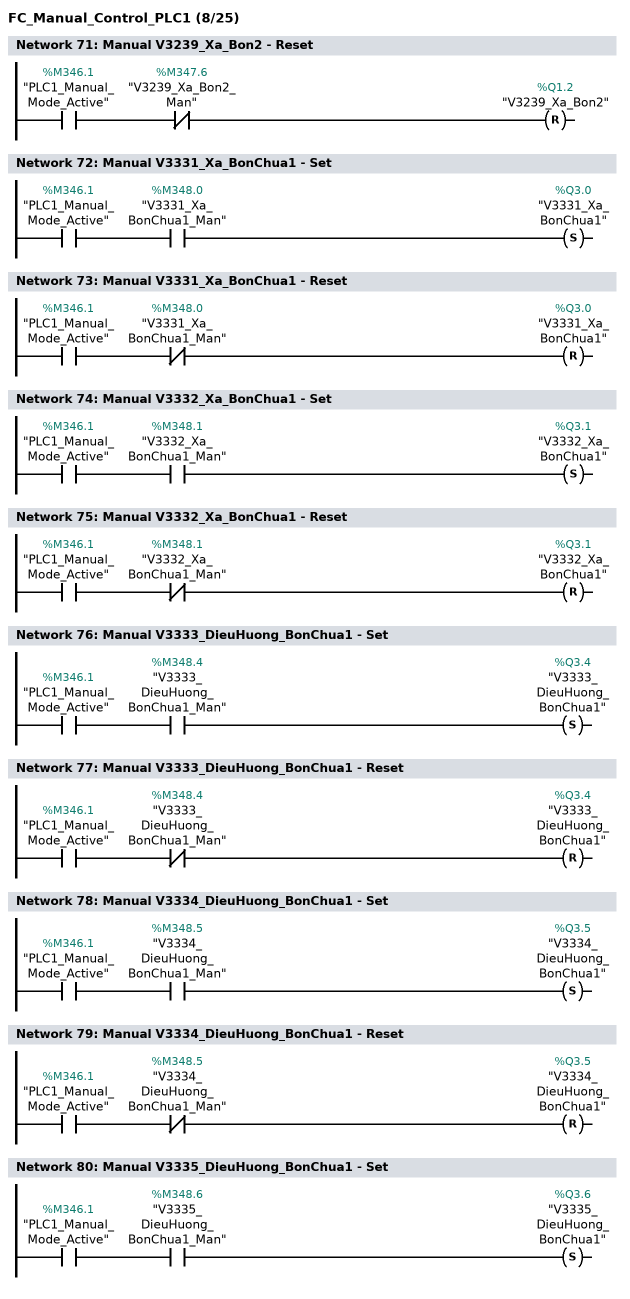
   RUNG wire#powerrail
      Contact( "PLC1_Manual_Mode_Active" )
      I_Contact( "V3239_Xa_Bon2_Man" )
      R_Coil( "V3239_Xa_Bon2" )
   END_RUNG
   // the same network as SCL:
   IF "PLC1_Manual_Mode_Active" AND NOT "V3239_Xa_Bon2_Man" THEN "V3239_Xa_Bon2" := FALSE; END_IF;
END_REGION

REGION Network 72: Manual V3331_Xa_BonChua1 - Set
   RUNG wire#powerrail
      Contact( "PLC1_Manual_Mode_Active" )
      Contact( "V3331_Xa_BonChua1_Man" )
      S_Coil( "V3331_Xa_BonChua1" )
   END_RUNG
   // the same network as SCL:
   IF "PLC1_Manual_Mode_Active" AND "V3331_Xa_BonChua1_Man" THEN "V3331_Xa_BonChua1" := TRUE; END_IF;
END_REGION

REGION Network 73: Manual V3331_Xa_BonChua1 - Reset
   RUNG wire#powerrail
      Contact( "PLC1_Manual_Mode_Active" )
      I_Contact( "V3331_Xa_BonChua1_Man" )
      R_Coil( "V3331_Xa_BonChua1" )
   END_RUNG
   // the same network as SCL:
   IF "PLC1_Manual_Mode_Active" AND NOT "V3331_Xa_BonChua1_Man" THEN "V3331_Xa_BonChua1" := FALSE; END_IF;
END_REGION

REGION Network 74: Manual V3332_Xa_BonChua1 - Set
   RUNG wire#powerrail
      Contact( "PLC1_Manual_Mode_Active" )
      Contact( "V3332_Xa_BonChua1_Man" )
      S_Coil( "V3332_Xa_BonChua1" )
   END_RUNG
   // the same network as SCL:
   IF "PLC1_Manual_Mode_Active" AND "V3332_Xa_BonChua1_Man" THEN "V3332_Xa_BonChua1" := TRUE; END_IF;
END_REGION

REGION Network 75: Manual V3332_Xa_BonChua1 - Reset
   RUNG wire#powerrail
      Contact( "PLC1_Manual_Mode_Active" )
      I_Contact( "V3332_Xa_BonChua1_Man" )
      R_Coil( "V3332_Xa_BonChua1" )
   END_RUNG
   // the same network as SCL:
   IF "PLC1_Manual_Mode_Active" AND NOT "V3332_Xa_BonChua1_Man" THEN "V3332_Xa_BonChua1" := FALSE; END_IF;
END_REGION

REGION Network 76: Manual V3333_DieuHuong_BonChua1 - Set
   RUNG wire#powerrail
      Contact( "PLC1_Manual_Mode_Active" )
      Contact( "V3333_DieuHuong_BonChua1_Man" )
      S_Coil( "V3333_DieuHuong_BonChua1" )
   END_RUNG
   // the same network as SCL:
   IF "PLC1_Manual_Mode_Active" AND "V3333_DieuHuong_BonChua1_Man" THEN
       "V3333_DieuHuong_BonChua1" := TRUE;
   END_IF;
END_REGION

REGION Network 77: Manual V3333_DieuHuong_BonChua1 - Reset
   RUNG wire#powerrail
      Contact( "PLC1_Manual_Mode_Active" )
      I_Contact( "V3333_DieuHuong_BonChua1_Man" )
      R_Coil( "V3333_DieuHuong_BonChua1" )
   END_RUNG
   // the same network as SCL:
   IF "PLC1_Manual_Mode_Active" AND NOT "V3333_DieuHuong_BonChua1_Man" THEN
       "V3333_DieuHuong_BonChua1" := FALSE;
   END_IF;
END_REGION

REGION Network 78: Manual V3334_DieuHuong_BonChua1 - Set
   RUNG wire#powerrail
      Contact( "PLC1_Manual_Mode_Active" )
      Contact( "V3334_DieuHuong_BonChua1_Man" )
      S_Coil( "V3334_DieuHuong_BonChua1" )
   END_RUNG
   // the same network as SCL:
   IF "PLC1_Manual_Mode_Active" AND "V3334_DieuHuong_BonChua1_Man" THEN
       "V3334_DieuHuong_BonChua1" := TRUE;
   END_IF;
END_REGION

REGION Network 79: Manual V3334_DieuHuong_BonChua1 - Reset
   RUNG wire#powerrail
      Contact( "PLC1_Manual_Mode_Active" )
      I_Contact( "V3334_DieuHuong_BonChua1_Man" )
      R_Coil( "V3334_DieuHuong_BonChua1" )
   END_RUNG
   // the same network as SCL:
   IF "PLC1_Manual_Mode_Active" AND NOT "V3334_DieuHuong_BonChua1_Man" THEN
       "V3334_DieuHuong_BonChua1" := FALSE;
   END_IF;
END_REGION

REGION Network 80: Manual V3335_DieuHuong_BonChua1 - Set
   RUNG wire#powerrail
      Contact( "PLC1_Manual_Mode_Active" )
      Contact( "V3335_DieuHuong_BonChua1_Man" )
      S_Coil( "V3335_DieuHuong_BonChua1" )
   END_RUNG
   // the same network as SCL:
   IF "PLC1_Manual_Mode_Active" AND "V3335_DieuHuong_BonChua1_Man" THEN
       "V3335_DieuHuong_BonChua1" := TRUE;
   END_IF;
END_REGION

REGION Network 81: Manual V3335_DieuHuong_BonChua1 - Reset
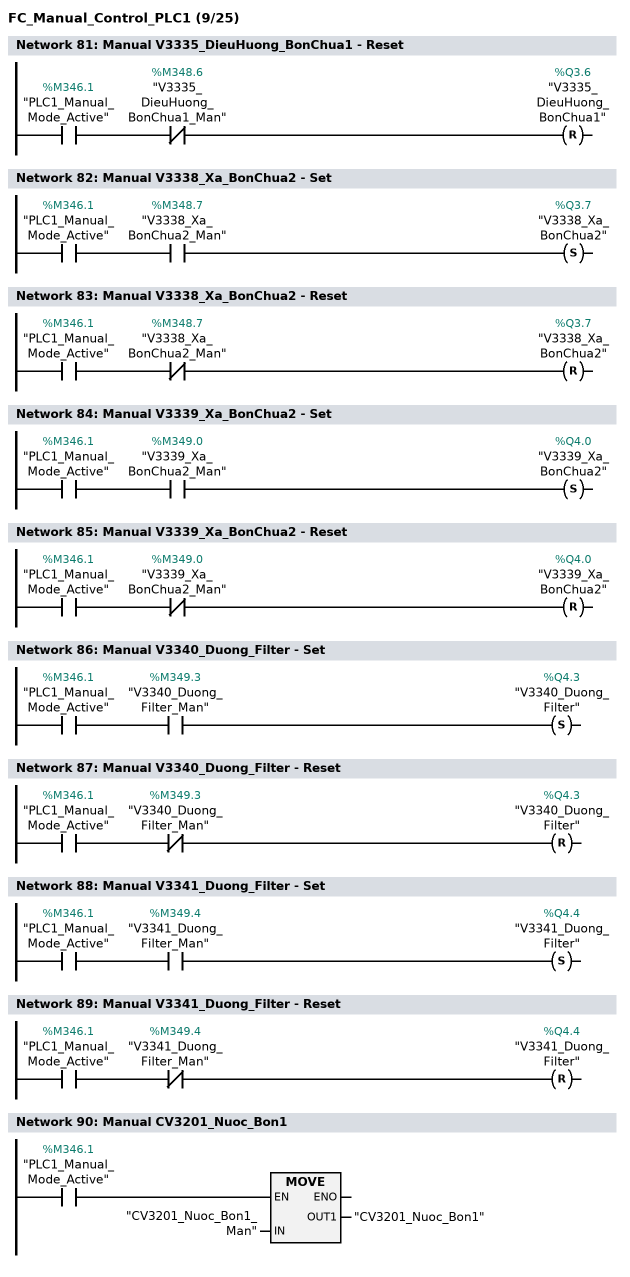
   RUNG wire#powerrail
      Contact( "PLC1_Manual_Mode_Active" )
      I_Contact( "V3335_DieuHuong_BonChua1_Man" )
      R_Coil( "V3335_DieuHuong_BonChua1" )
   END_RUNG
   // the same network as SCL:
   IF "PLC1_Manual_Mode_Active" AND NOT "V3335_DieuHuong_BonChua1_Man" THEN
       "V3335_DieuHuong_BonChua1" := FALSE;
   END_IF;
END_REGION

REGION Network 82: Manual V3338_Xa_BonChua2 - Set
   RUNG wire#powerrail
      Contact( "PLC1_Manual_Mode_Active" )
      Contact( "V3338_Xa_BonChua2_Man" )
      S_Coil( "V3338_Xa_BonChua2" )
   END_RUNG
   // the same network as SCL:
   IF "PLC1_Manual_Mode_Active" AND "V3338_Xa_BonChua2_Man" THEN "V3338_Xa_BonChua2" := TRUE; END_IF;
END_REGION

REGION Network 83: Manual V3338_Xa_BonChua2 - Reset
   RUNG wire#powerrail
      Contact( "PLC1_Manual_Mode_Active" )
      I_Contact( "V3338_Xa_BonChua2_Man" )
      R_Coil( "V3338_Xa_BonChua2" )
   END_RUNG
   // the same network as SCL:
   IF "PLC1_Manual_Mode_Active" AND NOT "V3338_Xa_BonChua2_Man" THEN "V3338_Xa_BonChua2" := FALSE; END_IF;
END_REGION

REGION Network 84: Manual V3339_Xa_BonChua2 - Set
   RUNG wire#powerrail
      Contact( "PLC1_Manual_Mode_Active" )
      Contact( "V3339_Xa_BonChua2_Man" )
      S_Coil( "V3339_Xa_BonChua2" )
   END_RUNG
   // the same network as SCL:
   IF "PLC1_Manual_Mode_Active" AND "V3339_Xa_BonChua2_Man" THEN "V3339_Xa_BonChua2" := TRUE; END_IF;
END_REGION

REGION Network 85: Manual V3339_Xa_BonChua2 - Reset
   RUNG wire#powerrail
      Contact( "PLC1_Manual_Mode_Active" )
      I_Contact( "V3339_Xa_BonChua2_Man" )
      R_Coil( "V3339_Xa_BonChua2" )
   END_RUNG
   // the same network as SCL:
   IF "PLC1_Manual_Mode_Active" AND NOT "V3339_Xa_BonChua2_Man" THEN "V3339_Xa_BonChua2" := FALSE; END_IF;
END_REGION

REGION Network 86: Manual V3340_Duong_Filter - Set
   RUNG wire#powerrail
      Contact( "PLC1_Manual_Mode_Active" )
      Contact( "V3340_Duong_Filter_Man" )
      S_Coil( "V3340_Duong_Filter" )
   END_RUNG
   // the same network as SCL:
   IF "PLC1_Manual_Mode_Active" AND "V3340_Duong_Filter_Man" THEN "V3340_Duong_Filter" := TRUE; END_IF;
END_REGION

REGION Network 87: Manual V3340_Duong_Filter - Reset
   RUNG wire#powerrail
      Contact( "PLC1_Manual_Mode_Active" )
      I_Contact( "V3340_Duong_Filter_Man" )
      R_Coil( "V3340_Duong_Filter" )
   END_RUNG
   // the same network as SCL:
   IF "PLC1_Manual_Mode_Active" AND NOT "V3340_Duong_Filter_Man" THEN "V3340_Duong_Filter" := FALSE; END_IF;
END_REGION

REGION Network 88: Manual V3341_Duong_Filter - Set
   RUNG wire#powerrail
      Contact( "PLC1_Manual_Mode_Active" )
      Contact( "V3341_Duong_Filter_Man" )
      S_Coil( "V3341_Duong_Filter" )
   END_RUNG
   // the same network as SCL:
   IF "PLC1_Manual_Mode_Active" AND "V3341_Duong_Filter_Man" THEN "V3341_Duong_Filter" := TRUE; END_IF;
END_REGION

REGION Network 89: Manual V3341_Duong_Filter - Reset
   RUNG wire#powerrail
      Contact( "PLC1_Manual_Mode_Active" )
      I_Contact( "V3341_Duong_Filter_Man" )
      R_Coil( "V3341_Duong_Filter" )
   END_RUNG
   // the same network as SCL:
   IF "PLC1_Manual_Mode_Active" AND NOT "V3341_Duong_Filter_Man" THEN "V3341_Duong_Filter" := FALSE; END_IF;
END_REGION

REGION Network 90: Manual CV3201_Nuoc_Bon1
   RUNG wire#powerrail
      Contact( "PLC1_Manual_Mode_Active" )
      { S7_GenerateENO := "TRUE" } Move(in := "CV3201_Nuoc_Bon1_Man", out1 => "CV3201_Nuoc_Bon1")
   END_RUNG
   // the same network as SCL:
   IF "PLC1_Manual_Mode_Active" THEN "CV3201_Nuoc_Bon1" := "CV3201_Nuoc_Bon1_Man"; END_IF;
END_REGION

REGION Network 91: Manual AGTR3260_Toc_Do_AO
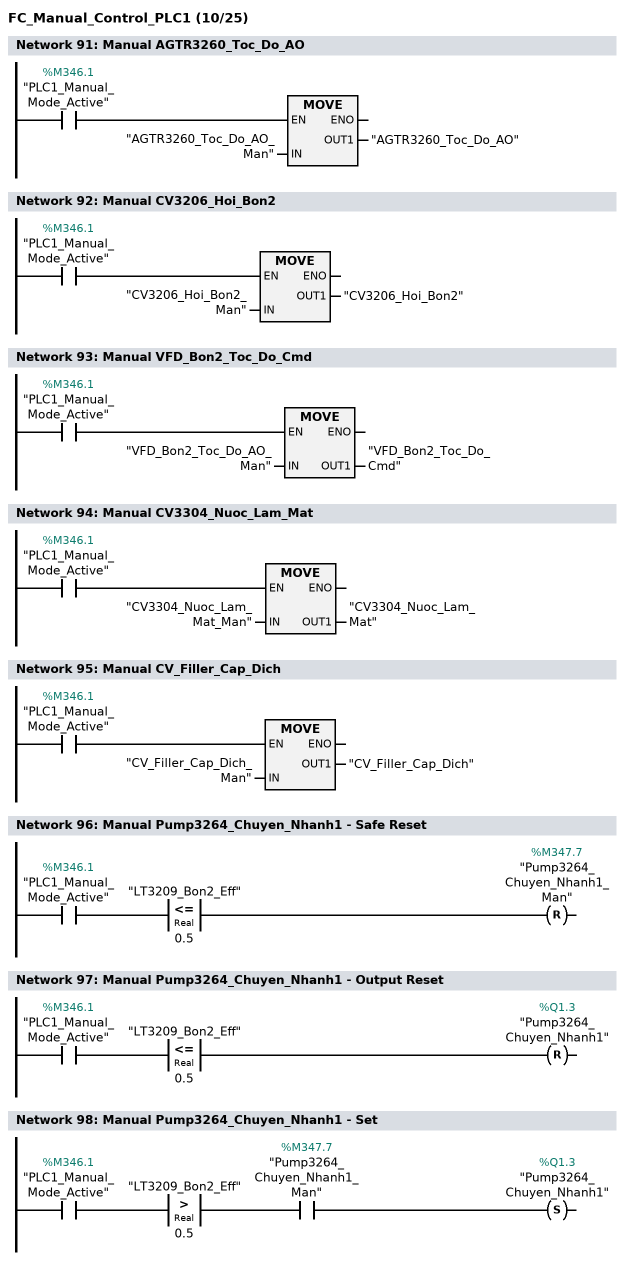
   RUNG wire#powerrail
      Contact( "PLC1_Manual_Mode_Active" )
      { S7_GenerateENO := "TRUE" } Move(in := "AGTR3260_Toc_Do_AO_Man", out1 => "AGTR3260_Toc_Do_AO")
   END_RUNG
   // the same network as SCL:
   IF "PLC1_Manual_Mode_Active" THEN "AGTR3260_Toc_Do_AO" := "AGTR3260_Toc_Do_AO_Man"; END_IF;
END_REGION

REGION Network 92: Manual CV3206_Hoi_Bon2
   RUNG wire#powerrail
      Contact( "PLC1_Manual_Mode_Active" )
      { S7_GenerateENO := "TRUE" } Move(in := "CV3206_Hoi_Bon2_Man", out1 => "CV3206_Hoi_Bon2")
   END_RUNG
   // the same network as SCL:
   IF "PLC1_Manual_Mode_Active" THEN "CV3206_Hoi_Bon2" := "CV3206_Hoi_Bon2_Man"; END_IF;
END_REGION

REGION Network 93: Manual VFD_Bon2_Toc_Do_Cmd
   RUNG wire#powerrail
      Contact( "PLC1_Manual_Mode_Active" )
      { S7_GenerateENO := "TRUE" } Move(in := "VFD_Bon2_Toc_Do_AO_Man", out1 => "VFD_Bon2_Toc_Do_Cmd")
   END_RUNG
   // the same network as SCL:
   IF "PLC1_Manual_Mode_Active" THEN "VFD_Bon2_Toc_Do_Cmd" := "VFD_Bon2_Toc_Do_AO_Man"; END_IF;
END_REGION

REGION Network 94: Manual CV3304_Nuoc_Lam_Mat
   RUNG wire#powerrail
      Contact( "PLC1_Manual_Mode_Active" )
      { S7_GenerateENO := "TRUE" } Move(in := "CV3304_Nuoc_Lam_Mat_Man", out1 => "CV3304_Nuoc_Lam_Mat")
   END_RUNG
   // the same network as SCL:
   IF "PLC1_Manual_Mode_Active" THEN "CV3304_Nuoc_Lam_Mat" := "CV3304_Nuoc_Lam_Mat_Man"; END_IF;
END_REGION

REGION Network 95: Manual CV_Filler_Cap_Dich
   RUNG wire#powerrail
      Contact( "PLC1_Manual_Mode_Active" )
      { S7_GenerateENO := "TRUE" } Move(in := "CV_Filler_Cap_Dich_Man", out1 => "CV_Filler_Cap_Dich")
   END_RUNG
   // the same network as SCL:
   IF "PLC1_Manual_Mode_Active" THEN "CV_Filler_Cap_Dich" := "CV_Filler_Cap_Dich_Man"; END_IF;
END_REGION

REGION Network 96: Manual Pump3264_Chuyen_Nhanh1 - Safe Reset
   RUNG wire#powerrail
      Contact( "PLC1_Manual_Mode_Active" )
      { S7_Templates := "SrcType := Real" } LE_Contact(in1 := "LT3209_Bon2_Eff", in2 := 0.5)
      R_Coil( "Pump3264_Chuyen_Nhanh1_Man" )
   END_RUNG
   // the same network as SCL:
   IF "PLC1_Manual_Mode_Active" AND ("LT3209_Bon2_Eff" <= 0.5) THEN
       "Pump3264_Chuyen_Nhanh1_Man" := FALSE;
   END_IF;
END_REGION

REGION Network 97: Manual Pump3264_Chuyen_Nhanh1 - Output Reset
   RUNG wire#powerrail
      Contact( "PLC1_Manual_Mode_Active" )
      { S7_Templates := "SrcType := Real" } LE_Contact(in1 := "LT3209_Bon2_Eff", in2 := 0.5)
      R_Coil( "Pump3264_Chuyen_Nhanh1" )
   END_RUNG
   // the same network as SCL:
   IF "PLC1_Manual_Mode_Active" AND ("LT3209_Bon2_Eff" <= 0.5) THEN
       "Pump3264_Chuyen_Nhanh1" := FALSE;
   END_IF;
END_REGION

REGION Network 98: Manual Pump3264_Chuyen_Nhanh1 - Set
   RUNG wire#powerrail
      Contact( "PLC1_Manual_Mode_Active" )
      { S7_Templates := "SrcType := Real" } GT_Contact(in1 := "LT3209_Bon2_Eff", in2 := 0.5)
      Contact( "Pump3264_Chuyen_Nhanh1_Man" )
      S_Coil( "Pump3264_Chuyen_Nhanh1" )
   END_RUNG
   // the same network as SCL:
   IF "PLC1_Manual_Mode_Active" AND ("LT3209_Bon2_Eff" > 0.5) AND "Pump3264_Chuyen_Nhanh1_Man" THEN
       "Pump3264_Chuyen_Nhanh1" := TRUE;
   END_IF;
END_REGION

REGION Network 99: Manual Pump3264_Chuyen_Nhanh1 - Reset
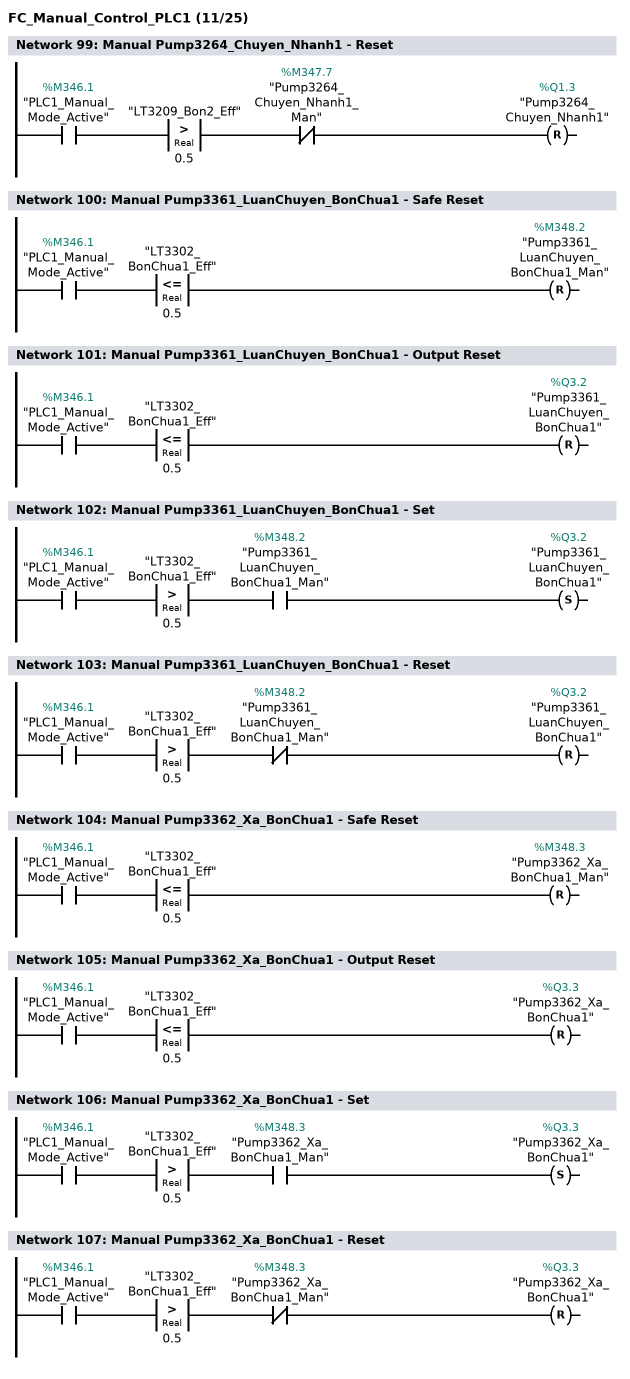
   RUNG wire#powerrail
      Contact( "PLC1_Manual_Mode_Active" )
      { S7_Templates := "SrcType := Real" } GT_Contact(in1 := "LT3209_Bon2_Eff", in2 := 0.5)
      I_Contact( "Pump3264_Chuyen_Nhanh1_Man" )
      R_Coil( "Pump3264_Chuyen_Nhanh1" )
   END_RUNG
   // the same network as SCL:
   IF "PLC1_Manual_Mode_Active" AND ("LT3209_Bon2_Eff" > 0.5) AND NOT "Pump3264_Chuyen_Nhanh1_Man" THEN
       "Pump3264_Chuyen_Nhanh1" := FALSE;
   END_IF;
END_REGION

REGION Network 100: Manual Pump3361_LuanChuyen_BonChua1 - Safe Reset
   RUNG wire#powerrail
      Contact( "PLC1_Manual_Mode_Active" )
      { S7_Templates := "SrcType := Real" } LE_Contact(in1 := "LT3302_BonChua1_Eff", in2 := 0.5)
      R_Coil( "Pump3361_LuanChuyen_BonChua1_Man" )
   END_RUNG
   // the same network as SCL:
   IF "PLC1_Manual_Mode_Active" AND ("LT3302_BonChua1_Eff" <= 0.5) THEN
       "Pump3361_LuanChuyen_BonChua1_Man" := FALSE;
   END_IF;
END_REGION

REGION Network 101: Manual Pump3361_LuanChuyen_BonChua1 - Output Reset
   RUNG wire#powerrail
      Contact( "PLC1_Manual_Mode_Active" )
      { S7_Templates := "SrcType := Real" } LE_Contact(in1 := "LT3302_BonChua1_Eff", in2 := 0.5)
      R_Coil( "Pump3361_LuanChuyen_BonChua1" )
   END_RUNG
   // the same network as SCL:
   IF "PLC1_Manual_Mode_Active" AND ("LT3302_BonChua1_Eff" <= 0.5) THEN
       "Pump3361_LuanChuyen_BonChua1" := FALSE;
   END_IF;
END_REGION

REGION Network 102: Manual Pump3361_LuanChuyen_BonChua1 - Set
   RUNG wire#powerrail
      Contact( "PLC1_Manual_Mode_Active" )
      { S7_Templates := "SrcType := Real" } GT_Contact(in1 := "LT3302_BonChua1_Eff", in2 := 0.5)
      Contact( "Pump3361_LuanChuyen_BonChua1_Man" )
      S_Coil( "Pump3361_LuanChuyen_BonChua1" )
   END_RUNG
   // the same network as SCL:
   IF "PLC1_Manual_Mode_Active" AND ("LT3302_BonChua1_Eff" > 0.5) AND "Pump3361_LuanChuyen_BonChua1_Man" THEN
       "Pump3361_LuanChuyen_BonChua1" := TRUE;
   END_IF;
END_REGION

REGION Network 103: Manual Pump3361_LuanChuyen_BonChua1 - Reset
   RUNG wire#powerrail
      Contact( "PLC1_Manual_Mode_Active" )
      { S7_Templates := "SrcType := Real" } GT_Contact(in1 := "LT3302_BonChua1_Eff", in2 := 0.5)
      I_Contact( "Pump3361_LuanChuyen_BonChua1_Man" )
      R_Coil( "Pump3361_LuanChuyen_BonChua1" )
   END_RUNG
   // the same network as SCL:
   IF "PLC1_Manual_Mode_Active" AND ("LT3302_BonChua1_Eff" > 0.5) AND NOT "Pump3361_LuanChuyen_BonChua1_Man" THEN
       "Pump3361_LuanChuyen_BonChua1" := FALSE;
   END_IF;
END_REGION

REGION Network 104: Manual Pump3362_Xa_BonChua1 - Safe Reset
   RUNG wire#powerrail
      Contact( "PLC1_Manual_Mode_Active" )
      { S7_Templates := "SrcType := Real" } LE_Contact(in1 := "LT3302_BonChua1_Eff", in2 := 0.5)
      R_Coil( "Pump3362_Xa_BonChua1_Man" )
   END_RUNG
   // the same network as SCL:
   IF "PLC1_Manual_Mode_Active" AND ("LT3302_BonChua1_Eff" <= 0.5) THEN
       "Pump3362_Xa_BonChua1_Man" := FALSE;
   END_IF;
END_REGION

REGION Network 105: Manual Pump3362_Xa_BonChua1 - Output Reset
   RUNG wire#powerrail
      Contact( "PLC1_Manual_Mode_Active" )
      { S7_Templates := "SrcType := Real" } LE_Contact(in1 := "LT3302_BonChua1_Eff", in2 := 0.5)
      R_Coil( "Pump3362_Xa_BonChua1" )
   END_RUNG
   // the same network as SCL:
   IF "PLC1_Manual_Mode_Active" AND ("LT3302_BonChua1_Eff" <= 0.5) THEN
       "Pump3362_Xa_BonChua1" := FALSE;
   END_IF;
END_REGION

REGION Network 106: Manual Pump3362_Xa_BonChua1 - Set
   RUNG wire#powerrail
      Contact( "PLC1_Manual_Mode_Active" )
      { S7_Templates := "SrcType := Real" } GT_Contact(in1 := "LT3302_BonChua1_Eff", in2 := 0.5)
      Contact( "Pump3362_Xa_BonChua1_Man" )
      S_Coil( "Pump3362_Xa_BonChua1" )
   END_RUNG
   // the same network as SCL:
   IF "PLC1_Manual_Mode_Active" AND ("LT3302_BonChua1_Eff" > 0.5) AND "Pump3362_Xa_BonChua1_Man" THEN
       "Pump3362_Xa_BonChua1" := TRUE;
   END_IF;
END_REGION

REGION Network 107: Manual Pump3362_Xa_BonChua1 - Reset
   RUNG wire#powerrail
      Contact( "PLC1_Manual_Mode_Active" )
      { S7_Templates := "SrcType := Real" } GT_Contact(in1 := "LT3302_BonChua1_Eff", in2 := 0.5)
      I_Contact( "Pump3362_Xa_BonChua1_Man" )
      R_Coil( "Pump3362_Xa_BonChua1" )
   END_RUNG
   // the same network as SCL:
   IF "PLC1_Manual_Mode_Active" AND ("LT3302_BonChua1_Eff" > 0.5) AND NOT "Pump3362_Xa_BonChua1_Man" THEN
       "Pump3362_Xa_BonChua1" := FALSE;
   END_IF;
END_REGION

REGION Network 108: Manual Pump3364_Filter - Safe Reset
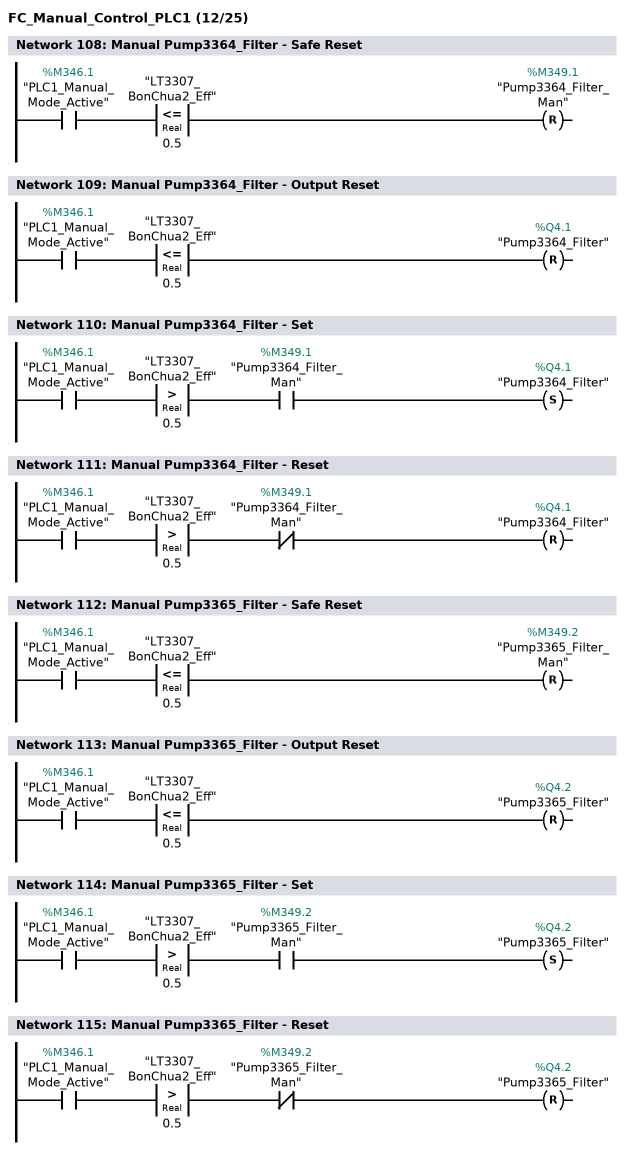
   RUNG wire#powerrail
      Contact( "PLC1_Manual_Mode_Active" )
      { S7_Templates := "SrcType := Real" } LE_Contact(in1 := "LT3307_BonChua2_Eff", in2 := 0.5)
      R_Coil( "Pump3364_Filter_Man" )
   END_RUNG
   // the same network as SCL:
   IF "PLC1_Manual_Mode_Active" AND ("LT3307_BonChua2_Eff" <= 0.5) THEN
       "Pump3364_Filter_Man" := FALSE;
   END_IF;
END_REGION

REGION Network 109: Manual Pump3364_Filter - Output Reset
   RUNG wire#powerrail
      Contact( "PLC1_Manual_Mode_Active" )
      { S7_Templates := "SrcType := Real" } LE_Contact(in1 := "LT3307_BonChua2_Eff", in2 := 0.5)
      R_Coil( "Pump3364_Filter" )
   END_RUNG
   // the same network as SCL:
   IF "PLC1_Manual_Mode_Active" AND ("LT3307_BonChua2_Eff" <= 0.5) THEN "Pump3364_Filter" := FALSE; END_IF;
END_REGION

REGION Network 110: Manual Pump3364_Filter - Set
   RUNG wire#powerrail
      Contact( "PLC1_Manual_Mode_Active" )
      { S7_Templates := "SrcType := Real" } GT_Contact(in1 := "LT3307_BonChua2_Eff", in2 := 0.5)
      Contact( "Pump3364_Filter_Man" )
      S_Coil( "Pump3364_Filter" )
   END_RUNG
   // the same network as SCL:
   IF "PLC1_Manual_Mode_Active" AND ("LT3307_BonChua2_Eff" > 0.5) AND "Pump3364_Filter_Man" THEN
       "Pump3364_Filter" := TRUE;
   END_IF;
END_REGION

REGION Network 111: Manual Pump3364_Filter - Reset
   RUNG wire#powerrail
      Contact( "PLC1_Manual_Mode_Active" )
      { S7_Templates := "SrcType := Real" } GT_Contact(in1 := "LT3307_BonChua2_Eff", in2 := 0.5)
      I_Contact( "Pump3364_Filter_Man" )
      R_Coil( "Pump3364_Filter" )
   END_RUNG
   // the same network as SCL:
   IF "PLC1_Manual_Mode_Active" AND ("LT3307_BonChua2_Eff" > 0.5) AND NOT "Pump3364_Filter_Man" THEN
       "Pump3364_Filter" := FALSE;
   END_IF;
END_REGION

REGION Network 112: Manual Pump3365_Filter - Safe Reset
   RUNG wire#powerrail
      Contact( "PLC1_Manual_Mode_Active" )
      { S7_Templates := "SrcType := Real" } LE_Contact(in1 := "LT3307_BonChua2_Eff", in2 := 0.5)
      R_Coil( "Pump3365_Filter_Man" )
   END_RUNG
   // the same network as SCL:
   IF "PLC1_Manual_Mode_Active" AND ("LT3307_BonChua2_Eff" <= 0.5) THEN
       "Pump3365_Filter_Man" := FALSE;
   END_IF;
END_REGION

REGION Network 113: Manual Pump3365_Filter - Output Reset
   RUNG wire#powerrail
      Contact( "PLC1_Manual_Mode_Active" )
      { S7_Templates := "SrcType := Real" } LE_Contact(in1 := "LT3307_BonChua2_Eff", in2 := 0.5)
      R_Coil( "Pump3365_Filter" )
   END_RUNG
   // the same network as SCL:
   IF "PLC1_Manual_Mode_Active" AND ("LT3307_BonChua2_Eff" <= 0.5) THEN "Pump3365_Filter" := FALSE; END_IF;
END_REGION

REGION Network 114: Manual Pump3365_Filter - Set
   RUNG wire#powerrail
      Contact( "PLC1_Manual_Mode_Active" )
      { S7_Templates := "SrcType := Real" } GT_Contact(in1 := "LT3307_BonChua2_Eff", in2 := 0.5)
      Contact( "Pump3365_Filter_Man" )
      S_Coil( "Pump3365_Filter" )
   END_RUNG
   // the same network as SCL:
   IF "PLC1_Manual_Mode_Active" AND ("LT3307_BonChua2_Eff" > 0.5) AND "Pump3365_Filter_Man" THEN
       "Pump3365_Filter" := TRUE;
   END_IF;
END_REGION

REGION Network 115: Manual Pump3365_Filter - Reset
   RUNG wire#powerrail
      Contact( "PLC1_Manual_Mode_Active" )
      { S7_Templates := "SrcType := Real" } GT_Contact(in1 := "LT3307_BonChua2_Eff", in2 := 0.5)
      I_Contact( "Pump3365_Filter_Man" )
      R_Coil( "Pump3365_Filter" )
   END_RUNG
   // the same network as SCL:
   IF "PLC1_Manual_Mode_Active" AND ("LT3307_BonChua2_Eff" > 0.5) AND NOT "Pump3365_Filter_Man" THEN
       "Pump3365_Filter" := FALSE;
   END_IF;
END_REGION

REGION Network 116: Safety override - Reset V3230_Nuoc_Bon1
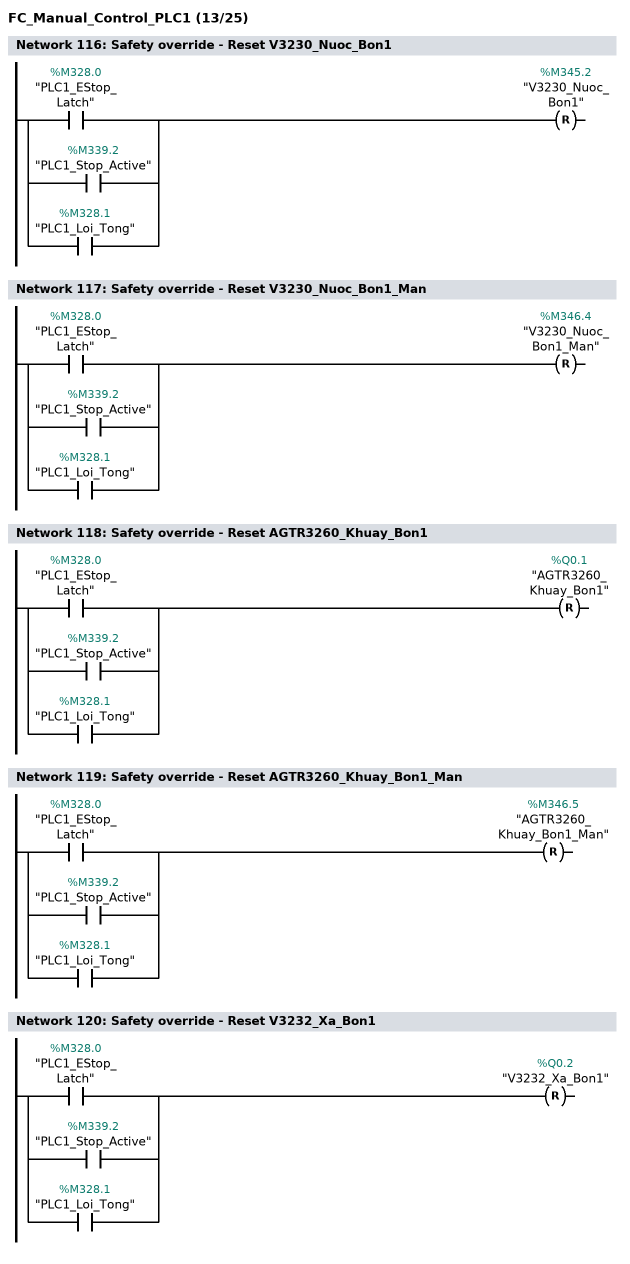
   RUNG wire#powerrail
      Contact( "PLC1_EStop_Latch" )
      wire#w1
      R_Coil( "V3230_Nuoc_Bon1" )
   END_RUNG
   RUNG wire#powerrail
      Contact( "PLC1_Stop_Active" )
   END_RUNG wire#w1
   RUNG wire#powerrail
      Contact( "PLC1_Loi_Tong" )
   END_RUNG wire#w1
   // the same network as SCL:
   IF "PLC1_EStop_Latch" OR "PLC1_Stop_Active" OR "PLC1_Loi_Tong" THEN "V3230_Nuoc_Bon1" := FALSE; END_IF;
END_REGION

REGION Network 117: Safety override - Reset V3230_Nuoc_Bon1_Man
   RUNG wire#powerrail
      Contact( "PLC1_EStop_Latch" )
      wire#w1
      R_Coil( "V3230_Nuoc_Bon1_Man" )
   END_RUNG
   RUNG wire#powerrail
      Contact( "PLC1_Stop_Active" )
   END_RUNG wire#w1
   RUNG wire#powerrail
      Contact( "PLC1_Loi_Tong" )
   END_RUNG wire#w1
   // the same network as SCL:
   IF "PLC1_EStop_Latch" OR "PLC1_Stop_Active" OR "PLC1_Loi_Tong" THEN
       "V3230_Nuoc_Bon1_Man" := FALSE;
   END_IF;
END_REGION

REGION Network 118: Safety override - Reset AGTR3260_Khuay_Bon1
   RUNG wire#powerrail
      Contact( "PLC1_EStop_Latch" )
      wire#w1
      R_Coil( "AGTR3260_Khuay_Bon1" )
   END_RUNG
   RUNG wire#powerrail
      Contact( "PLC1_Stop_Active" )
   END_RUNG wire#w1
   RUNG wire#powerrail
      Contact( "PLC1_Loi_Tong" )
   END_RUNG wire#w1
   // the same network as SCL:
   IF "PLC1_EStop_Latch" OR "PLC1_Stop_Active" OR "PLC1_Loi_Tong" THEN
       "AGTR3260_Khuay_Bon1" := FALSE;
   END_IF;
END_REGION

REGION Network 119: Safety override - Reset AGTR3260_Khuay_Bon1_Man
   RUNG wire#powerrail
      Contact( "PLC1_EStop_Latch" )
      wire#w1
      R_Coil( "AGTR3260_Khuay_Bon1_Man" )
   END_RUNG
   RUNG wire#powerrail
      Contact( "PLC1_Stop_Active" )
   END_RUNG wire#w1
   RUNG wire#powerrail
      Contact( "PLC1_Loi_Tong" )
   END_RUNG wire#w1
   // the same network as SCL:
   IF "PLC1_EStop_Latch" OR "PLC1_Stop_Active" OR "PLC1_Loi_Tong" THEN
       "AGTR3260_Khuay_Bon1_Man" := FALSE;
   END_IF;
END_REGION

REGION Network 120: Safety override - Reset V3232_Xa_Bon1
   RUNG wire#powerrail
      Contact( "PLC1_EStop_Latch" )
      wire#w1
      R_Coil( "V3232_Xa_Bon1" )
   END_RUNG
   RUNG wire#powerrail
      Contact( "PLC1_Stop_Active" )
   END_RUNG wire#w1
   RUNG wire#powerrail
      Contact( "PLC1_Loi_Tong" )
   END_RUNG wire#w1
   // the same network as SCL:
   IF "PLC1_EStop_Latch" OR "PLC1_Stop_Active" OR "PLC1_Loi_Tong" THEN "V3232_Xa_Bon1" := FALSE; END_IF;
END_REGION

REGION Network 121: Safety override - Reset V3232_Xa_Bon1_Man
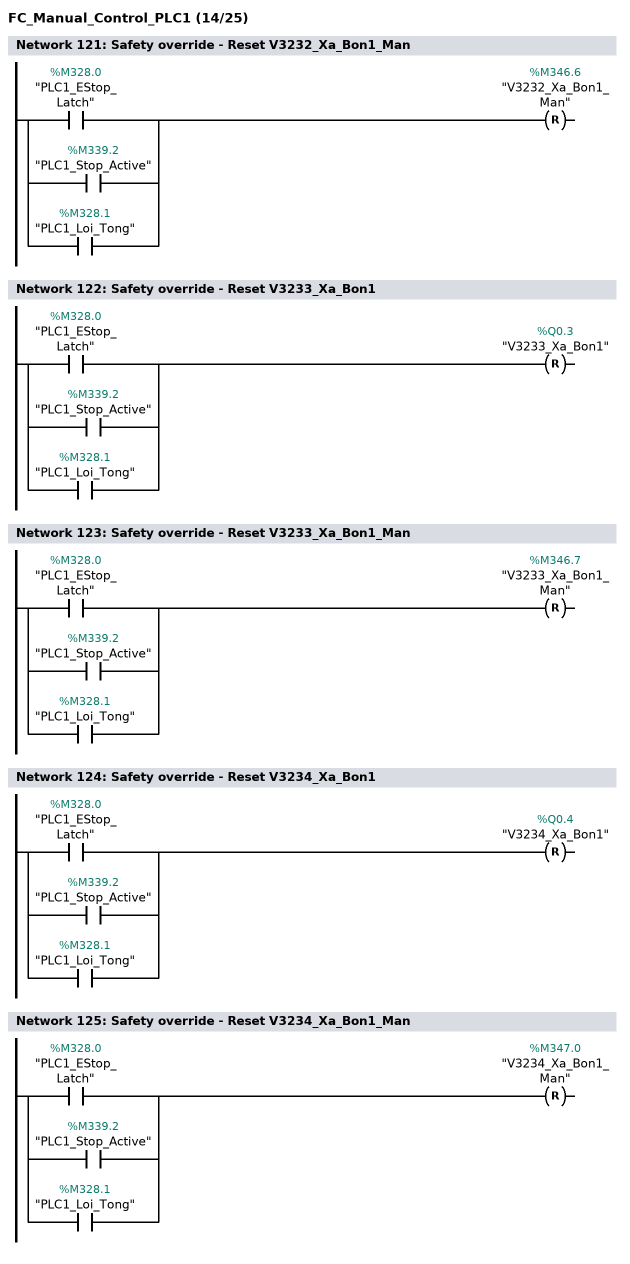
   RUNG wire#powerrail
      Contact( "PLC1_EStop_Latch" )
      wire#w1
      R_Coil( "V3232_Xa_Bon1_Man" )
   END_RUNG
   RUNG wire#powerrail
      Contact( "PLC1_Stop_Active" )
   END_RUNG wire#w1
   RUNG wire#powerrail
      Contact( "PLC1_Loi_Tong" )
   END_RUNG wire#w1
   // the same network as SCL:
   IF "PLC1_EStop_Latch" OR "PLC1_Stop_Active" OR "PLC1_Loi_Tong" THEN "V3232_Xa_Bon1_Man" := FALSE; END_IF;
END_REGION

REGION Network 122: Safety override - Reset V3233_Xa_Bon1
   RUNG wire#powerrail
      Contact( "PLC1_EStop_Latch" )
      wire#w1
      R_Coil( "V3233_Xa_Bon1" )
   END_RUNG
   RUNG wire#powerrail
      Contact( "PLC1_Stop_Active" )
   END_RUNG wire#w1
   RUNG wire#powerrail
      Contact( "PLC1_Loi_Tong" )
   END_RUNG wire#w1
   // the same network as SCL:
   IF "PLC1_EStop_Latch" OR "PLC1_Stop_Active" OR "PLC1_Loi_Tong" THEN "V3233_Xa_Bon1" := FALSE; END_IF;
END_REGION

REGION Network 123: Safety override - Reset V3233_Xa_Bon1_Man
   RUNG wire#powerrail
      Contact( "PLC1_EStop_Latch" )
      wire#w1
      R_Coil( "V3233_Xa_Bon1_Man" )
   END_RUNG
   RUNG wire#powerrail
      Contact( "PLC1_Stop_Active" )
   END_RUNG wire#w1
   RUNG wire#powerrail
      Contact( "PLC1_Loi_Tong" )
   END_RUNG wire#w1
   // the same network as SCL:
   IF "PLC1_EStop_Latch" OR "PLC1_Stop_Active" OR "PLC1_Loi_Tong" THEN "V3233_Xa_Bon1_Man" := FALSE; END_IF;
END_REGION

REGION Network 124: Safety override - Reset V3234_Xa_Bon1
   RUNG wire#powerrail
      Contact( "PLC1_EStop_Latch" )
      wire#w1
      R_Coil( "V3234_Xa_Bon1" )
   END_RUNG
   RUNG wire#powerrail
      Contact( "PLC1_Stop_Active" )
   END_RUNG wire#w1
   RUNG wire#powerrail
      Contact( "PLC1_Loi_Tong" )
   END_RUNG wire#w1
   // the same network as SCL:
   IF "PLC1_EStop_Latch" OR "PLC1_Stop_Active" OR "PLC1_Loi_Tong" THEN "V3234_Xa_Bon1" := FALSE; END_IF;
END_REGION

REGION Network 125: Safety override - Reset V3234_Xa_Bon1_Man
   RUNG wire#powerrail
      Contact( "PLC1_EStop_Latch" )
      wire#w1
      R_Coil( "V3234_Xa_Bon1_Man" )
   END_RUNG
   RUNG wire#powerrail
      Contact( "PLC1_Stop_Active" )
   END_RUNG wire#w1
   RUNG wire#powerrail
      Contact( "PLC1_Loi_Tong" )
   END_RUNG wire#w1
   // the same network as SCL:
   IF "PLC1_EStop_Latch" OR "PLC1_Stop_Active" OR "PLC1_Loi_Tong" THEN "V3234_Xa_Bon1_Man" := FALSE; END_IF;
END_REGION

REGION Network 126: Safety override - Reset V3235_Nuoc_Bon2
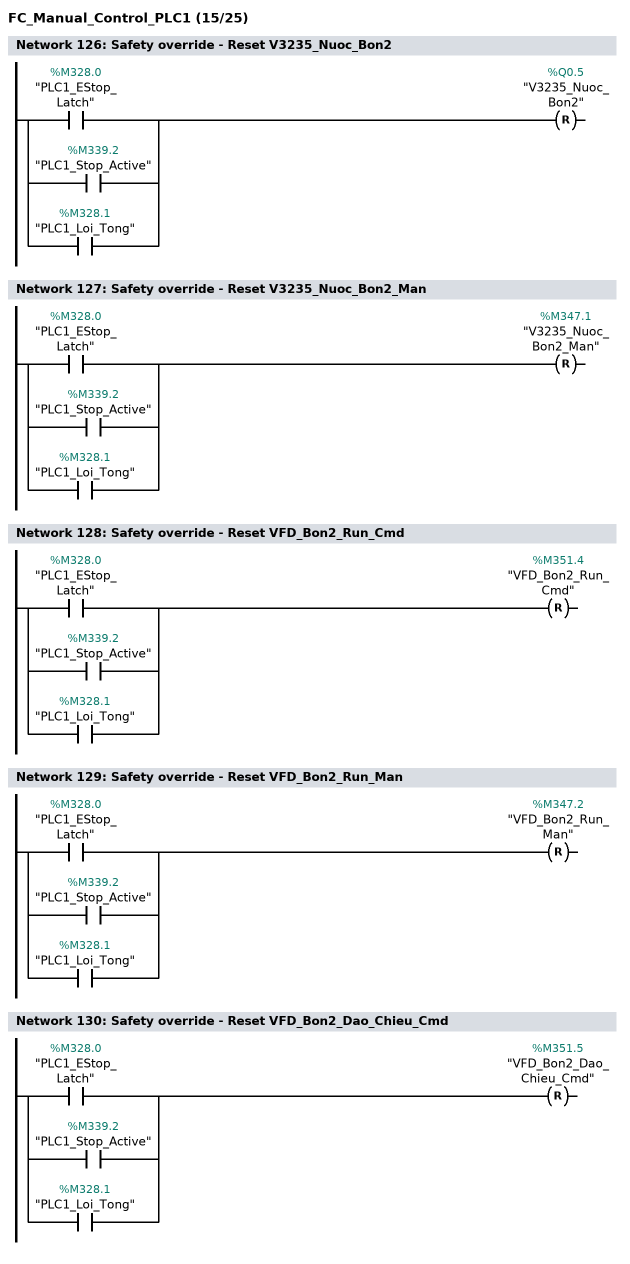
   RUNG wire#powerrail
      Contact( "PLC1_EStop_Latch" )
      wire#w1
      R_Coil( "V3235_Nuoc_Bon2" )
   END_RUNG
   RUNG wire#powerrail
      Contact( "PLC1_Stop_Active" )
   END_RUNG wire#w1
   RUNG wire#powerrail
      Contact( "PLC1_Loi_Tong" )
   END_RUNG wire#w1
   // the same network as SCL:
   IF "PLC1_EStop_Latch" OR "PLC1_Stop_Active" OR "PLC1_Loi_Tong" THEN "V3235_Nuoc_Bon2" := FALSE; END_IF;
END_REGION

REGION Network 127: Safety override - Reset V3235_Nuoc_Bon2_Man
   RUNG wire#powerrail
      Contact( "PLC1_EStop_Latch" )
      wire#w1
      R_Coil( "V3235_Nuoc_Bon2_Man" )
   END_RUNG
   RUNG wire#powerrail
      Contact( "PLC1_Stop_Active" )
   END_RUNG wire#w1
   RUNG wire#powerrail
      Contact( "PLC1_Loi_Tong" )
   END_RUNG wire#w1
   // the same network as SCL:
   IF "PLC1_EStop_Latch" OR "PLC1_Stop_Active" OR "PLC1_Loi_Tong" THEN
       "V3235_Nuoc_Bon2_Man" := FALSE;
   END_IF;
END_REGION

REGION Network 128: Safety override - Reset VFD_Bon2_Run_Cmd
   RUNG wire#powerrail
      Contact( "PLC1_EStop_Latch" )
      wire#w1
      R_Coil( "VFD_Bon2_Run_Cmd" )
   END_RUNG
   RUNG wire#powerrail
      Contact( "PLC1_Stop_Active" )
   END_RUNG wire#w1
   RUNG wire#powerrail
      Contact( "PLC1_Loi_Tong" )
   END_RUNG wire#w1
   // the same network as SCL:
   IF "PLC1_EStop_Latch" OR "PLC1_Stop_Active" OR "PLC1_Loi_Tong" THEN "VFD_Bon2_Run_Cmd" := FALSE; END_IF;
END_REGION

REGION Network 129: Safety override - Reset VFD_Bon2_Run_Man
   RUNG wire#powerrail
      Contact( "PLC1_EStop_Latch" )
      wire#w1
      R_Coil( "VFD_Bon2_Run_Man" )
   END_RUNG
   RUNG wire#powerrail
      Contact( "PLC1_Stop_Active" )
   END_RUNG wire#w1
   RUNG wire#powerrail
      Contact( "PLC1_Loi_Tong" )
   END_RUNG wire#w1
   // the same network as SCL:
   IF "PLC1_EStop_Latch" OR "PLC1_Stop_Active" OR "PLC1_Loi_Tong" THEN "VFD_Bon2_Run_Man" := FALSE; END_IF;
END_REGION

REGION Network 130: Safety override - Reset VFD_Bon2_Dao_Chieu_Cmd
   RUNG wire#powerrail
      Contact( "PLC1_EStop_Latch" )
      wire#w1
      R_Coil( "VFD_Bon2_Dao_Chieu_Cmd" )
   END_RUNG
   RUNG wire#powerrail
      Contact( "PLC1_Stop_Active" )
   END_RUNG wire#w1
   RUNG wire#powerrail
      Contact( "PLC1_Loi_Tong" )
   END_RUNG wire#w1
   // the same network as SCL:
   IF "PLC1_EStop_Latch" OR "PLC1_Stop_Active" OR "PLC1_Loi_Tong" THEN
       "VFD_Bon2_Dao_Chieu_Cmd" := FALSE;
   END_IF;
END_REGION

REGION Network 131: Safety override - Reset VFD_Bon2_Dao_Chieu_Man
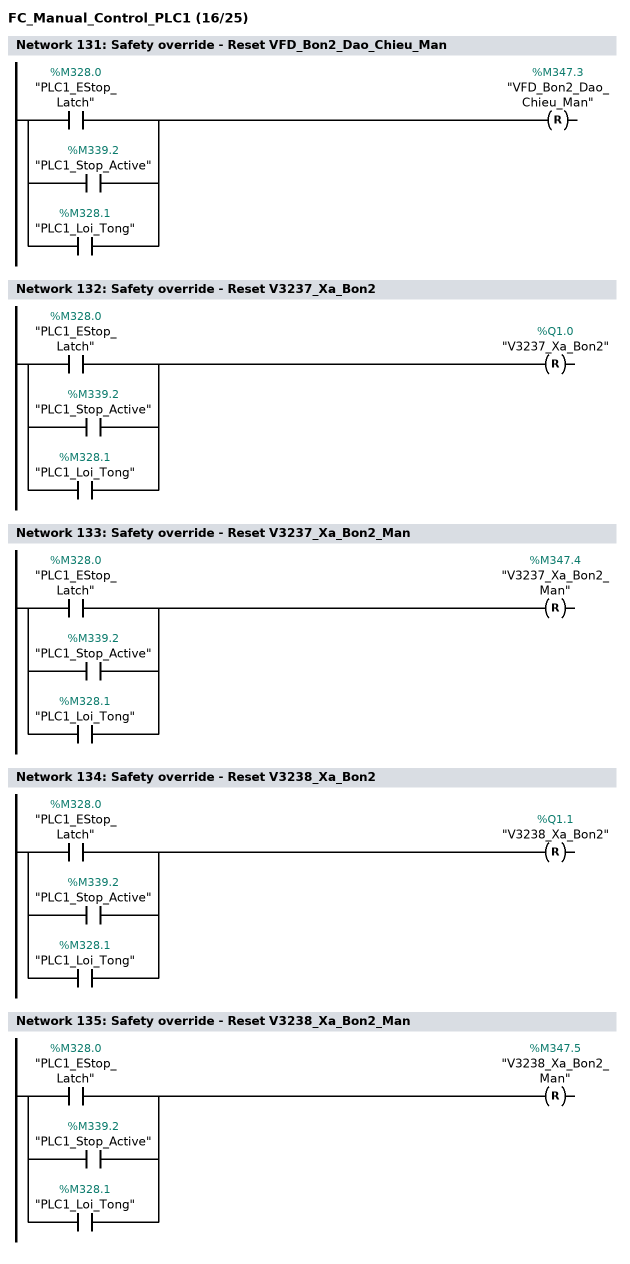
   RUNG wire#powerrail
      Contact( "PLC1_EStop_Latch" )
      wire#w1
      R_Coil( "VFD_Bon2_Dao_Chieu_Man" )
   END_RUNG
   RUNG wire#powerrail
      Contact( "PLC1_Stop_Active" )
   END_RUNG wire#w1
   RUNG wire#powerrail
      Contact( "PLC1_Loi_Tong" )
   END_RUNG wire#w1
   // the same network as SCL:
   IF "PLC1_EStop_Latch" OR "PLC1_Stop_Active" OR "PLC1_Loi_Tong" THEN
       "VFD_Bon2_Dao_Chieu_Man" := FALSE;
   END_IF;
END_REGION

REGION Network 132: Safety override - Reset V3237_Xa_Bon2
   RUNG wire#powerrail
      Contact( "PLC1_EStop_Latch" )
      wire#w1
      R_Coil( "V3237_Xa_Bon2" )
   END_RUNG
   RUNG wire#powerrail
      Contact( "PLC1_Stop_Active" )
   END_RUNG wire#w1
   RUNG wire#powerrail
      Contact( "PLC1_Loi_Tong" )
   END_RUNG wire#w1
   // the same network as SCL:
   IF "PLC1_EStop_Latch" OR "PLC1_Stop_Active" OR "PLC1_Loi_Tong" THEN "V3237_Xa_Bon2" := FALSE; END_IF;
END_REGION

REGION Network 133: Safety override - Reset V3237_Xa_Bon2_Man
   RUNG wire#powerrail
      Contact( "PLC1_EStop_Latch" )
      wire#w1
      R_Coil( "V3237_Xa_Bon2_Man" )
   END_RUNG
   RUNG wire#powerrail
      Contact( "PLC1_Stop_Active" )
   END_RUNG wire#w1
   RUNG wire#powerrail
      Contact( "PLC1_Loi_Tong" )
   END_RUNG wire#w1
   // the same network as SCL:
   IF "PLC1_EStop_Latch" OR "PLC1_Stop_Active" OR "PLC1_Loi_Tong" THEN "V3237_Xa_Bon2_Man" := FALSE; END_IF;
END_REGION

REGION Network 134: Safety override - Reset V3238_Xa_Bon2
   RUNG wire#powerrail
      Contact( "PLC1_EStop_Latch" )
      wire#w1
      R_Coil( "V3238_Xa_Bon2" )
   END_RUNG
   RUNG wire#powerrail
      Contact( "PLC1_Stop_Active" )
   END_RUNG wire#w1
   RUNG wire#powerrail
      Contact( "PLC1_Loi_Tong" )
   END_RUNG wire#w1
   // the same network as SCL:
   IF "PLC1_EStop_Latch" OR "PLC1_Stop_Active" OR "PLC1_Loi_Tong" THEN "V3238_Xa_Bon2" := FALSE; END_IF;
END_REGION

REGION Network 135: Safety override - Reset V3238_Xa_Bon2_Man
   RUNG wire#powerrail
      Contact( "PLC1_EStop_Latch" )
      wire#w1
      R_Coil( "V3238_Xa_Bon2_Man" )
   END_RUNG
   RUNG wire#powerrail
      Contact( "PLC1_Stop_Active" )
   END_RUNG wire#w1
   RUNG wire#powerrail
      Contact( "PLC1_Loi_Tong" )
   END_RUNG wire#w1
   // the same network as SCL:
   IF "PLC1_EStop_Latch" OR "PLC1_Stop_Active" OR "PLC1_Loi_Tong" THEN "V3238_Xa_Bon2_Man" := FALSE; END_IF;
END_REGION

REGION Network 136: Safety override - Reset V3239_Xa_Bon2
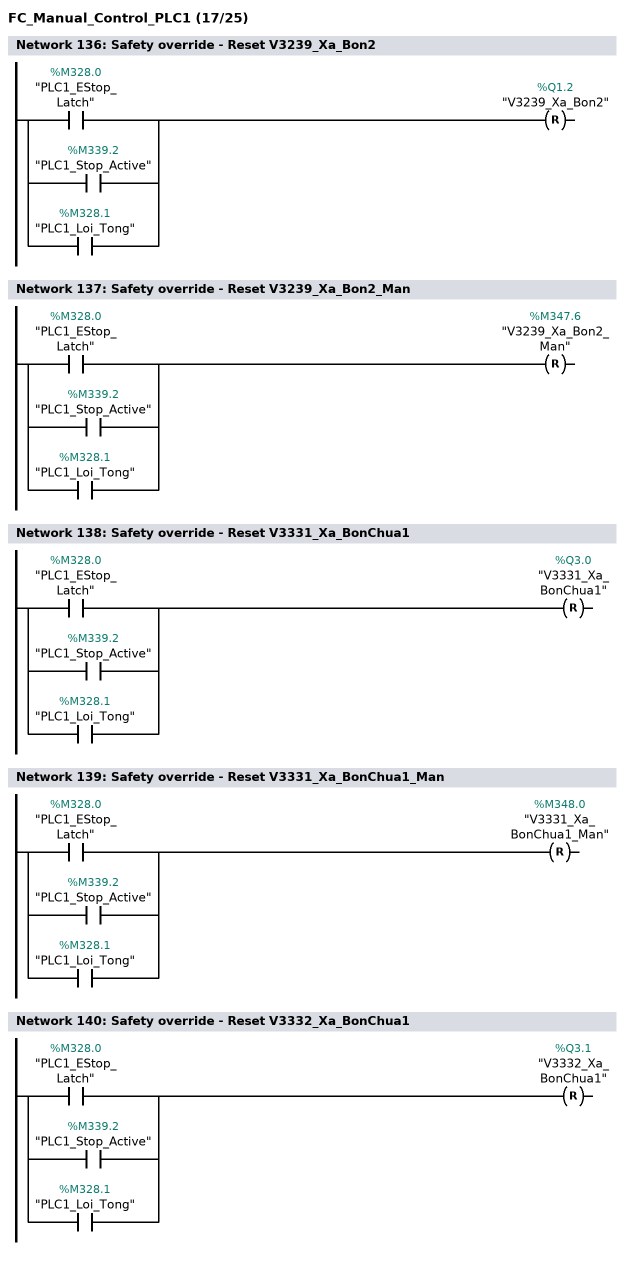
   RUNG wire#powerrail
      Contact( "PLC1_EStop_Latch" )
      wire#w1
      R_Coil( "V3239_Xa_Bon2" )
   END_RUNG
   RUNG wire#powerrail
      Contact( "PLC1_Stop_Active" )
   END_RUNG wire#w1
   RUNG wire#powerrail
      Contact( "PLC1_Loi_Tong" )
   END_RUNG wire#w1
   // the same network as SCL:
   IF "PLC1_EStop_Latch" OR "PLC1_Stop_Active" OR "PLC1_Loi_Tong" THEN "V3239_Xa_Bon2" := FALSE; END_IF;
END_REGION

REGION Network 137: Safety override - Reset V3239_Xa_Bon2_Man
   RUNG wire#powerrail
      Contact( "PLC1_EStop_Latch" )
      wire#w1
      R_Coil( "V3239_Xa_Bon2_Man" )
   END_RUNG
   RUNG wire#powerrail
      Contact( "PLC1_Stop_Active" )
   END_RUNG wire#w1
   RUNG wire#powerrail
      Contact( "PLC1_Loi_Tong" )
   END_RUNG wire#w1
   // the same network as SCL:
   IF "PLC1_EStop_Latch" OR "PLC1_Stop_Active" OR "PLC1_Loi_Tong" THEN "V3239_Xa_Bon2_Man" := FALSE; END_IF;
END_REGION

REGION Network 138: Safety override - Reset V3331_Xa_BonChua1
   RUNG wire#powerrail
      Contact( "PLC1_EStop_Latch" )
      wire#w1
      R_Coil( "V3331_Xa_BonChua1" )
   END_RUNG
   RUNG wire#powerrail
      Contact( "PLC1_Stop_Active" )
   END_RUNG wire#w1
   RUNG wire#powerrail
      Contact( "PLC1_Loi_Tong" )
   END_RUNG wire#w1
   // the same network as SCL:
   IF "PLC1_EStop_Latch" OR "PLC1_Stop_Active" OR "PLC1_Loi_Tong" THEN "V3331_Xa_BonChua1" := FALSE; END_IF;
END_REGION

REGION Network 139: Safety override - Reset V3331_Xa_BonChua1_Man
   RUNG wire#powerrail
      Contact( "PLC1_EStop_Latch" )
      wire#w1
      R_Coil( "V3331_Xa_BonChua1_Man" )
   END_RUNG
   RUNG wire#powerrail
      Contact( "PLC1_Stop_Active" )
   END_RUNG wire#w1
   RUNG wire#powerrail
      Contact( "PLC1_Loi_Tong" )
   END_RUNG wire#w1
   // the same network as SCL:
   IF "PLC1_EStop_Latch" OR "PLC1_Stop_Active" OR "PLC1_Loi_Tong" THEN
       "V3331_Xa_BonChua1_Man" := FALSE;
   END_IF;
END_REGION

REGION Network 140: Safety override - Reset V3332_Xa_BonChua1
   RUNG wire#powerrail
      Contact( "PLC1_EStop_Latch" )
      wire#w1
      R_Coil( "V3332_Xa_BonChua1" )
   END_RUNG
   RUNG wire#powerrail
      Contact( "PLC1_Stop_Active" )
   END_RUNG wire#w1
   RUNG wire#powerrail
      Contact( "PLC1_Loi_Tong" )
   END_RUNG wire#w1
   // the same network as SCL:
   IF "PLC1_EStop_Latch" OR "PLC1_Stop_Active" OR "PLC1_Loi_Tong" THEN "V3332_Xa_BonChua1" := FALSE; END_IF;
END_REGION

REGION Network 141: Safety override - Reset V3332_Xa_BonChua1_Man
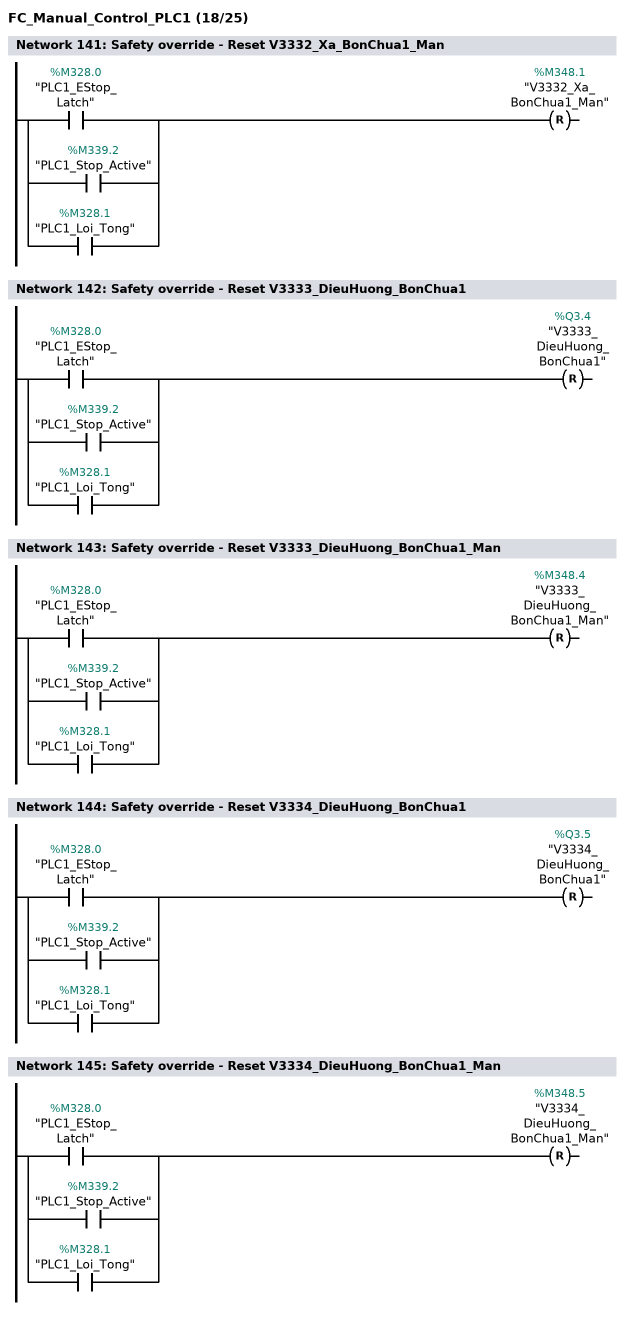
   RUNG wire#powerrail
      Contact( "PLC1_EStop_Latch" )
      wire#w1
      R_Coil( "V3332_Xa_BonChua1_Man" )
   END_RUNG
   RUNG wire#powerrail
      Contact( "PLC1_Stop_Active" )
   END_RUNG wire#w1
   RUNG wire#powerrail
      Contact( "PLC1_Loi_Tong" )
   END_RUNG wire#w1
   // the same network as SCL:
   IF "PLC1_EStop_Latch" OR "PLC1_Stop_Active" OR "PLC1_Loi_Tong" THEN
       "V3332_Xa_BonChua1_Man" := FALSE;
   END_IF;
END_REGION

REGION Network 142: Safety override - Reset V3333_DieuHuong_BonChua1
   RUNG wire#powerrail
      Contact( "PLC1_EStop_Latch" )
      wire#w1
      R_Coil( "V3333_DieuHuong_BonChua1" )
   END_RUNG
   RUNG wire#powerrail
      Contact( "PLC1_Stop_Active" )
   END_RUNG wire#w1
   RUNG wire#powerrail
      Contact( "PLC1_Loi_Tong" )
   END_RUNG wire#w1
   // the same network as SCL:
   IF "PLC1_EStop_Latch" OR "PLC1_Stop_Active" OR "PLC1_Loi_Tong" THEN
       "V3333_DieuHuong_BonChua1" := FALSE;
   END_IF;
END_REGION

REGION Network 143: Safety override - Reset V3333_DieuHuong_BonChua1_Man
   RUNG wire#powerrail
      Contact( "PLC1_EStop_Latch" )
      wire#w1
      R_Coil( "V3333_DieuHuong_BonChua1_Man" )
   END_RUNG
   RUNG wire#powerrail
      Contact( "PLC1_Stop_Active" )
   END_RUNG wire#w1
   RUNG wire#powerrail
      Contact( "PLC1_Loi_Tong" )
   END_RUNG wire#w1
   // the same network as SCL:
   IF "PLC1_EStop_Latch" OR "PLC1_Stop_Active" OR "PLC1_Loi_Tong" THEN
       "V3333_DieuHuong_BonChua1_Man" := FALSE;
   END_IF;
END_REGION

REGION Network 144: Safety override - Reset V3334_DieuHuong_BonChua1
   RUNG wire#powerrail
      Contact( "PLC1_EStop_Latch" )
      wire#w1
      R_Coil( "V3334_DieuHuong_BonChua1" )
   END_RUNG
   RUNG wire#powerrail
      Contact( "PLC1_Stop_Active" )
   END_RUNG wire#w1
   RUNG wire#powerrail
      Contact( "PLC1_Loi_Tong" )
   END_RUNG wire#w1
   // the same network as SCL:
   IF "PLC1_EStop_Latch" OR "PLC1_Stop_Active" OR "PLC1_Loi_Tong" THEN
       "V3334_DieuHuong_BonChua1" := FALSE;
   END_IF;
END_REGION

REGION Network 145: Safety override - Reset V3334_DieuHuong_BonChua1_Man
   RUNG wire#powerrail
      Contact( "PLC1_EStop_Latch" )
      wire#w1
      R_Coil( "V3334_DieuHuong_BonChua1_Man" )
   END_RUNG
   RUNG wire#powerrail
      Contact( "PLC1_Stop_Active" )
   END_RUNG wire#w1
   RUNG wire#powerrail
      Contact( "PLC1_Loi_Tong" )
   END_RUNG wire#w1
   // the same network as SCL:
   IF "PLC1_EStop_Latch" OR "PLC1_Stop_Active" OR "PLC1_Loi_Tong" THEN
       "V3334_DieuHuong_BonChua1_Man" := FALSE;
   END_IF;
END_REGION

REGION Network 146: Safety override - Reset V3335_DieuHuong_BonChua1
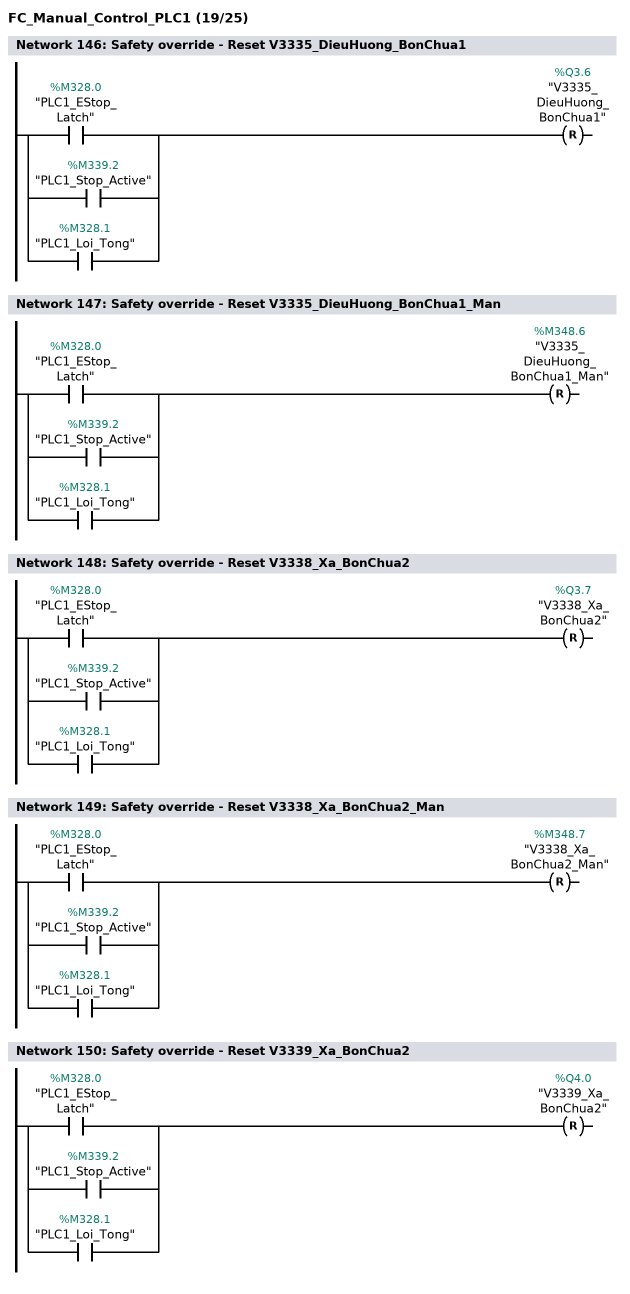
   RUNG wire#powerrail
      Contact( "PLC1_EStop_Latch" )
      wire#w1
      R_Coil( "V3335_DieuHuong_BonChua1" )
   END_RUNG
   RUNG wire#powerrail
      Contact( "PLC1_Stop_Active" )
   END_RUNG wire#w1
   RUNG wire#powerrail
      Contact( "PLC1_Loi_Tong" )
   END_RUNG wire#w1
   // the same network as SCL:
   IF "PLC1_EStop_Latch" OR "PLC1_Stop_Active" OR "PLC1_Loi_Tong" THEN
       "V3335_DieuHuong_BonChua1" := FALSE;
   END_IF;
END_REGION

REGION Network 147: Safety override - Reset V3335_DieuHuong_BonChua1_Man
   RUNG wire#powerrail
      Contact( "PLC1_EStop_Latch" )
      wire#w1
      R_Coil( "V3335_DieuHuong_BonChua1_Man" )
   END_RUNG
   RUNG wire#powerrail
      Contact( "PLC1_Stop_Active" )
   END_RUNG wire#w1
   RUNG wire#powerrail
      Contact( "PLC1_Loi_Tong" )
   END_RUNG wire#w1
   // the same network as SCL:
   IF "PLC1_EStop_Latch" OR "PLC1_Stop_Active" OR "PLC1_Loi_Tong" THEN
       "V3335_DieuHuong_BonChua1_Man" := FALSE;
   END_IF;
END_REGION

REGION Network 148: Safety override - Reset V3338_Xa_BonChua2
   RUNG wire#powerrail
      Contact( "PLC1_EStop_Latch" )
      wire#w1
      R_Coil( "V3338_Xa_BonChua2" )
   END_RUNG
   RUNG wire#powerrail
      Contact( "PLC1_Stop_Active" )
   END_RUNG wire#w1
   RUNG wire#powerrail
      Contact( "PLC1_Loi_Tong" )
   END_RUNG wire#w1
   // the same network as SCL:
   IF "PLC1_EStop_Latch" OR "PLC1_Stop_Active" OR "PLC1_Loi_Tong" THEN "V3338_Xa_BonChua2" := FALSE; END_IF;
END_REGION

REGION Network 149: Safety override - Reset V3338_Xa_BonChua2_Man
   RUNG wire#powerrail
      Contact( "PLC1_EStop_Latch" )
      wire#w1
      R_Coil( "V3338_Xa_BonChua2_Man" )
   END_RUNG
   RUNG wire#powerrail
      Contact( "PLC1_Stop_Active" )
   END_RUNG wire#w1
   RUNG wire#powerrail
      Contact( "PLC1_Loi_Tong" )
   END_RUNG wire#w1
   // the same network as SCL:
   IF "PLC1_EStop_Latch" OR "PLC1_Stop_Active" OR "PLC1_Loi_Tong" THEN
       "V3338_Xa_BonChua2_Man" := FALSE;
   END_IF;
END_REGION

REGION Network 150: Safety override - Reset V3339_Xa_BonChua2
   RUNG wire#powerrail
      Contact( "PLC1_EStop_Latch" )
      wire#w1
      R_Coil( "V3339_Xa_BonChua2" )
   END_RUNG
   RUNG wire#powerrail
      Contact( "PLC1_Stop_Active" )
   END_RUNG wire#w1
   RUNG wire#powerrail
      Contact( "PLC1_Loi_Tong" )
   END_RUNG wire#w1
   // the same network as SCL:
   IF "PLC1_EStop_Latch" OR "PLC1_Stop_Active" OR "PLC1_Loi_Tong" THEN "V3339_Xa_BonChua2" := FALSE; END_IF;
END_REGION

REGION Network 151: Safety override - Reset V3339_Xa_BonChua2_Man
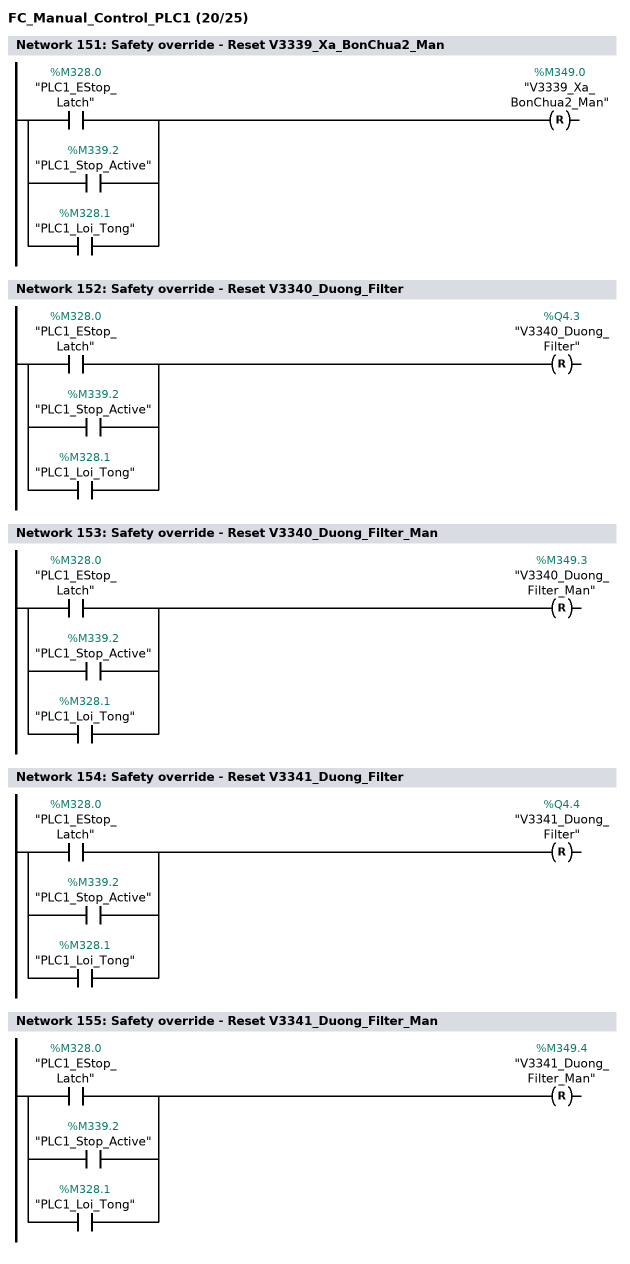
   RUNG wire#powerrail
      Contact( "PLC1_EStop_Latch" )
      wire#w1
      R_Coil( "V3339_Xa_BonChua2_Man" )
   END_RUNG
   RUNG wire#powerrail
      Contact( "PLC1_Stop_Active" )
   END_RUNG wire#w1
   RUNG wire#powerrail
      Contact( "PLC1_Loi_Tong" )
   END_RUNG wire#w1
   // the same network as SCL:
   IF "PLC1_EStop_Latch" OR "PLC1_Stop_Active" OR "PLC1_Loi_Tong" THEN
       "V3339_Xa_BonChua2_Man" := FALSE;
   END_IF;
END_REGION

REGION Network 152: Safety override - Reset V3340_Duong_Filter
   RUNG wire#powerrail
      Contact( "PLC1_EStop_Latch" )
      wire#w1
      R_Coil( "V3340_Duong_Filter" )
   END_RUNG
   RUNG wire#powerrail
      Contact( "PLC1_Stop_Active" )
   END_RUNG wire#w1
   RUNG wire#powerrail
      Contact( "PLC1_Loi_Tong" )
   END_RUNG wire#w1
   // the same network as SCL:
   IF "PLC1_EStop_Latch" OR "PLC1_Stop_Active" OR "PLC1_Loi_Tong" THEN "V3340_Duong_Filter" := FALSE; END_IF;
END_REGION

REGION Network 153: Safety override - Reset V3340_Duong_Filter_Man
   RUNG wire#powerrail
      Contact( "PLC1_EStop_Latch" )
      wire#w1
      R_Coil( "V3340_Duong_Filter_Man" )
   END_RUNG
   RUNG wire#powerrail
      Contact( "PLC1_Stop_Active" )
   END_RUNG wire#w1
   RUNG wire#powerrail
      Contact( "PLC1_Loi_Tong" )
   END_RUNG wire#w1
   // the same network as SCL:
   IF "PLC1_EStop_Latch" OR "PLC1_Stop_Active" OR "PLC1_Loi_Tong" THEN
       "V3340_Duong_Filter_Man" := FALSE;
   END_IF;
END_REGION

REGION Network 154: Safety override - Reset V3341_Duong_Filter
   RUNG wire#powerrail
      Contact( "PLC1_EStop_Latch" )
      wire#w1
      R_Coil( "V3341_Duong_Filter" )
   END_RUNG
   RUNG wire#powerrail
      Contact( "PLC1_Stop_Active" )
   END_RUNG wire#w1
   RUNG wire#powerrail
      Contact( "PLC1_Loi_Tong" )
   END_RUNG wire#w1
   // the same network as SCL:
   IF "PLC1_EStop_Latch" OR "PLC1_Stop_Active" OR "PLC1_Loi_Tong" THEN "V3341_Duong_Filter" := FALSE; END_IF;
END_REGION

REGION Network 155: Safety override - Reset V3341_Duong_Filter_Man
   RUNG wire#powerrail
      Contact( "PLC1_EStop_Latch" )
      wire#w1
      R_Coil( "V3341_Duong_Filter_Man" )
   END_RUNG
   RUNG wire#powerrail
      Contact( "PLC1_Stop_Active" )
   END_RUNG wire#w1
   RUNG wire#powerrail
      Contact( "PLC1_Loi_Tong" )
   END_RUNG wire#w1
   // the same network as SCL:
   IF "PLC1_EStop_Latch" OR "PLC1_Stop_Active" OR "PLC1_Loi_Tong" THEN
       "V3341_Duong_Filter_Man" := FALSE;
   END_IF;
END_REGION

REGION Network 156: Safety override - Reset Pump3264_Chuyen_Nhanh1
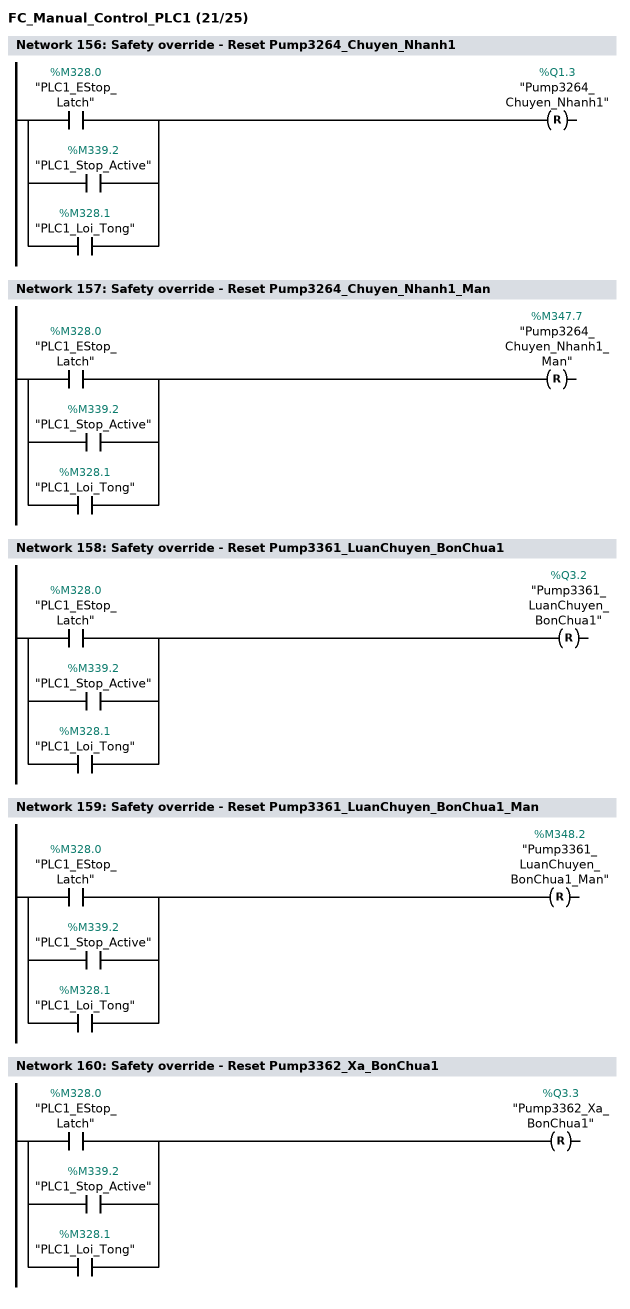
   RUNG wire#powerrail
      Contact( "PLC1_EStop_Latch" )
      wire#w1
      R_Coil( "Pump3264_Chuyen_Nhanh1" )
   END_RUNG
   RUNG wire#powerrail
      Contact( "PLC1_Stop_Active" )
   END_RUNG wire#w1
   RUNG wire#powerrail
      Contact( "PLC1_Loi_Tong" )
   END_RUNG wire#w1
   // the same network as SCL:
   IF "PLC1_EStop_Latch" OR "PLC1_Stop_Active" OR "PLC1_Loi_Tong" THEN
       "Pump3264_Chuyen_Nhanh1" := FALSE;
   END_IF;
END_REGION

REGION Network 157: Safety override - Reset Pump3264_Chuyen_Nhanh1_Man
   RUNG wire#powerrail
      Contact( "PLC1_EStop_Latch" )
      wire#w1
      R_Coil( "Pump3264_Chuyen_Nhanh1_Man" )
   END_RUNG
   RUNG wire#powerrail
      Contact( "PLC1_Stop_Active" )
   END_RUNG wire#w1
   RUNG wire#powerrail
      Contact( "PLC1_Loi_Tong" )
   END_RUNG wire#w1
   // the same network as SCL:
   IF "PLC1_EStop_Latch" OR "PLC1_Stop_Active" OR "PLC1_Loi_Tong" THEN
       "Pump3264_Chuyen_Nhanh1_Man" := FALSE;
   END_IF;
END_REGION

REGION Network 158: Safety override - Reset Pump3361_LuanChuyen_BonChua1
   RUNG wire#powerrail
      Contact( "PLC1_EStop_Latch" )
      wire#w1
      R_Coil( "Pump3361_LuanChuyen_BonChua1" )
   END_RUNG
   RUNG wire#powerrail
      Contact( "PLC1_Stop_Active" )
   END_RUNG wire#w1
   RUNG wire#powerrail
      Contact( "PLC1_Loi_Tong" )
   END_RUNG wire#w1
   // the same network as SCL:
   IF "PLC1_EStop_Latch" OR "PLC1_Stop_Active" OR "PLC1_Loi_Tong" THEN
       "Pump3361_LuanChuyen_BonChua1" := FALSE;
   END_IF;
END_REGION

REGION Network 159: Safety override - Reset Pump3361_LuanChuyen_BonChua1_Man
   RUNG wire#powerrail
      Contact( "PLC1_EStop_Latch" )
      wire#w1
      R_Coil( "Pump3361_LuanChuyen_BonChua1_Man" )
   END_RUNG
   RUNG wire#powerrail
      Contact( "PLC1_Stop_Active" )
   END_RUNG wire#w1
   RUNG wire#powerrail
      Contact( "PLC1_Loi_Tong" )
   END_RUNG wire#w1
   // the same network as SCL:
   IF "PLC1_EStop_Latch" OR "PLC1_Stop_Active" OR "PLC1_Loi_Tong" THEN
       "Pump3361_LuanChuyen_BonChua1_Man" := FALSE;
   END_IF;
END_REGION

REGION Network 160: Safety override - Reset Pump3362_Xa_BonChua1
   RUNG wire#powerrail
      Contact( "PLC1_EStop_Latch" )
      wire#w1
      R_Coil( "Pump3362_Xa_BonChua1" )
   END_RUNG
   RUNG wire#powerrail
      Contact( "PLC1_Stop_Active" )
   END_RUNG wire#w1
   RUNG wire#powerrail
      Contact( "PLC1_Loi_Tong" )
   END_RUNG wire#w1
   // the same network as SCL:
   IF "PLC1_EStop_Latch" OR "PLC1_Stop_Active" OR "PLC1_Loi_Tong" THEN
       "Pump3362_Xa_BonChua1" := FALSE;
   END_IF;
END_REGION

REGION Network 161: Safety override - Reset Pump3362_Xa_BonChua1_Man
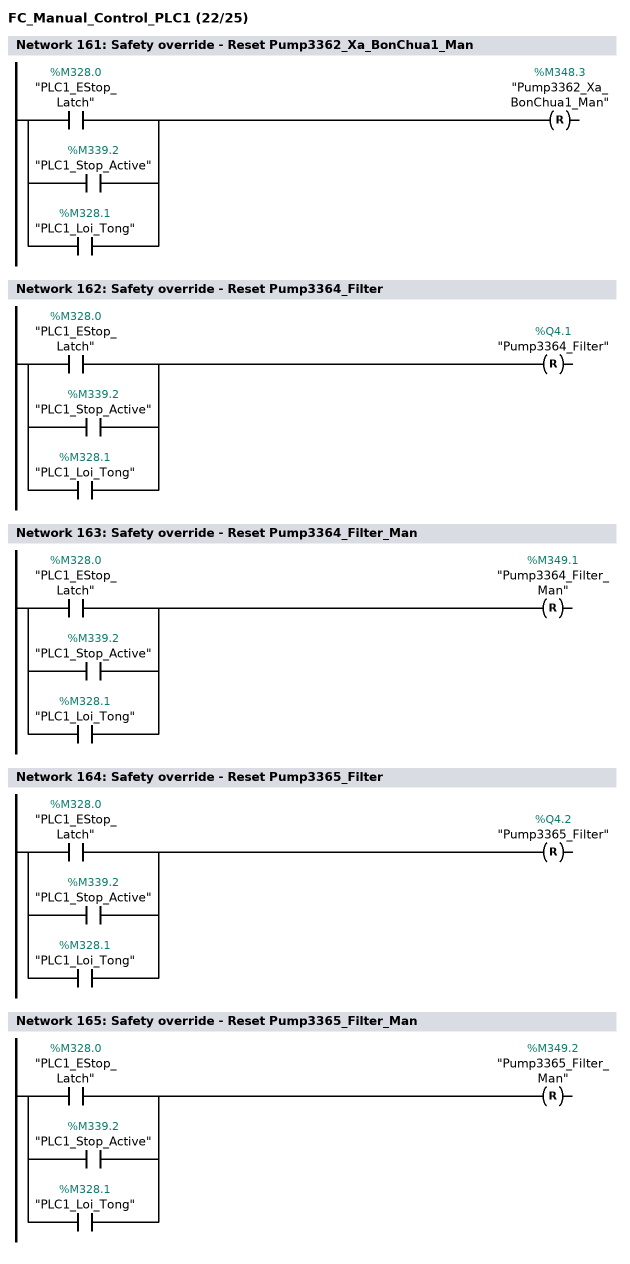
   RUNG wire#powerrail
      Contact( "PLC1_EStop_Latch" )
      wire#w1
      R_Coil( "Pump3362_Xa_BonChua1_Man" )
   END_RUNG
   RUNG wire#powerrail
      Contact( "PLC1_Stop_Active" )
   END_RUNG wire#w1
   RUNG wire#powerrail
      Contact( "PLC1_Loi_Tong" )
   END_RUNG wire#w1
   // the same network as SCL:
   IF "PLC1_EStop_Latch" OR "PLC1_Stop_Active" OR "PLC1_Loi_Tong" THEN
       "Pump3362_Xa_BonChua1_Man" := FALSE;
   END_IF;
END_REGION

REGION Network 162: Safety override - Reset Pump3364_Filter
   RUNG wire#powerrail
      Contact( "PLC1_EStop_Latch" )
      wire#w1
      R_Coil( "Pump3364_Filter" )
   END_RUNG
   RUNG wire#powerrail
      Contact( "PLC1_Stop_Active" )
   END_RUNG wire#w1
   RUNG wire#powerrail
      Contact( "PLC1_Loi_Tong" )
   END_RUNG wire#w1
   // the same network as SCL:
   IF "PLC1_EStop_Latch" OR "PLC1_Stop_Active" OR "PLC1_Loi_Tong" THEN "Pump3364_Filter" := FALSE; END_IF;
END_REGION

REGION Network 163: Safety override - Reset Pump3364_Filter_Man
   RUNG wire#powerrail
      Contact( "PLC1_EStop_Latch" )
      wire#w1
      R_Coil( "Pump3364_Filter_Man" )
   END_RUNG
   RUNG wire#powerrail
      Contact( "PLC1_Stop_Active" )
   END_RUNG wire#w1
   RUNG wire#powerrail
      Contact( "PLC1_Loi_Tong" )
   END_RUNG wire#w1
   // the same network as SCL:
   IF "PLC1_EStop_Latch" OR "PLC1_Stop_Active" OR "PLC1_Loi_Tong" THEN
       "Pump3364_Filter_Man" := FALSE;
   END_IF;
END_REGION

REGION Network 164: Safety override - Reset Pump3365_Filter
   RUNG wire#powerrail
      Contact( "PLC1_EStop_Latch" )
      wire#w1
      R_Coil( "Pump3365_Filter" )
   END_RUNG
   RUNG wire#powerrail
      Contact( "PLC1_Stop_Active" )
   END_RUNG wire#w1
   RUNG wire#powerrail
      Contact( "PLC1_Loi_Tong" )
   END_RUNG wire#w1
   // the same network as SCL:
   IF "PLC1_EStop_Latch" OR "PLC1_Stop_Active" OR "PLC1_Loi_Tong" THEN "Pump3365_Filter" := FALSE; END_IF;
END_REGION

REGION Network 165: Safety override - Reset Pump3365_Filter_Man
   RUNG wire#powerrail
      Contact( "PLC1_EStop_Latch" )
      wire#w1
      R_Coil( "Pump3365_Filter_Man" )
   END_RUNG
   RUNG wire#powerrail
      Contact( "PLC1_Stop_Active" )
   END_RUNG wire#w1
   RUNG wire#powerrail
      Contact( "PLC1_Loi_Tong" )
   END_RUNG wire#w1
   // the same network as SCL:
   IF "PLC1_EStop_Latch" OR "PLC1_Stop_Active" OR "PLC1_Loi_Tong" THEN
       "Pump3365_Filter_Man" := FALSE;
   END_IF;
END_REGION

REGION Network 166: Safety override - Clear CV3201_Nuoc_Bon1
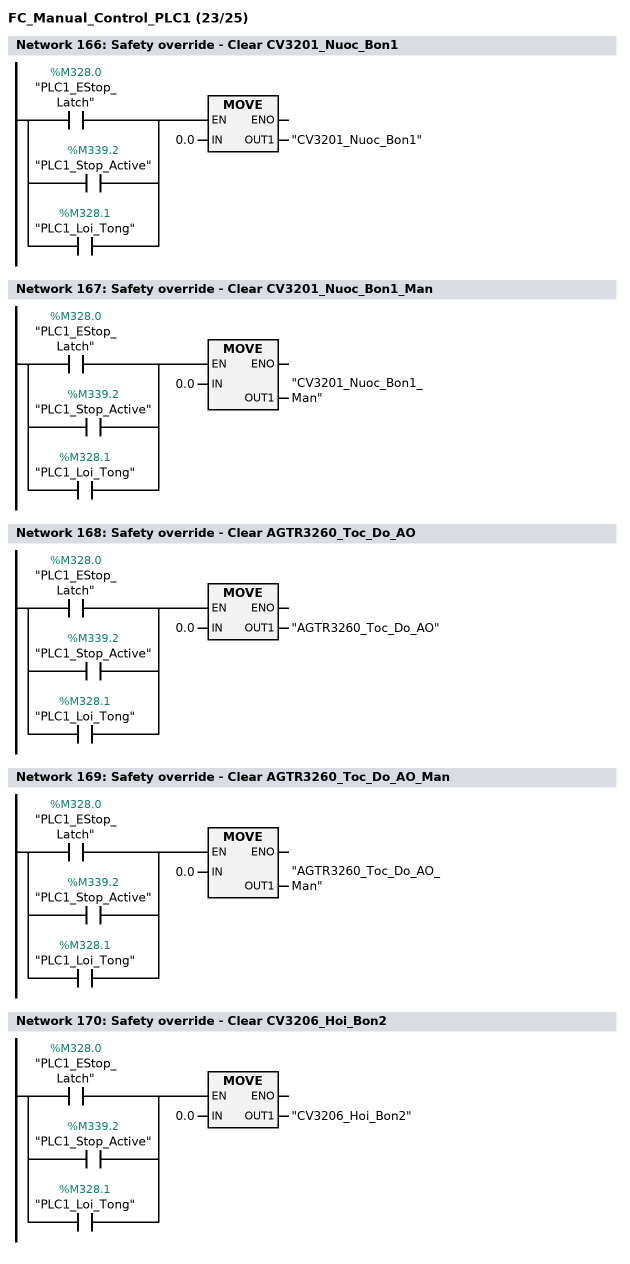
   RUNG wire#powerrail
      Contact( "PLC1_EStop_Latch" )
      wire#w1
      { S7_GenerateENO := "TRUE" } Move(in := 0.0, out1 => "CV3201_Nuoc_Bon1")
   END_RUNG
   RUNG wire#powerrail
      Contact( "PLC1_Stop_Active" )
   END_RUNG wire#w1
   RUNG wire#powerrail
      Contact( "PLC1_Loi_Tong" )
   END_RUNG wire#w1
   // the same network as SCL:
   IF "PLC1_EStop_Latch" OR "PLC1_Stop_Active" OR "PLC1_Loi_Tong" THEN "CV3201_Nuoc_Bon1" := 0.0; END_IF;
END_REGION

REGION Network 167: Safety override - Clear CV3201_Nuoc_Bon1_Man
   RUNG wire#powerrail
      Contact( "PLC1_EStop_Latch" )
      wire#w1
      { S7_GenerateENO := "TRUE" } Move(in := 0.0, out1 => "CV3201_Nuoc_Bon1_Man")
   END_RUNG
   RUNG wire#powerrail
      Contact( "PLC1_Stop_Active" )
   END_RUNG wire#w1
   RUNG wire#powerrail
      Contact( "PLC1_Loi_Tong" )
   END_RUNG wire#w1
   // the same network as SCL:
   IF "PLC1_EStop_Latch" OR "PLC1_Stop_Active" OR "PLC1_Loi_Tong" THEN "CV3201_Nuoc_Bon1_Man" := 0.0; END_IF;
END_REGION

REGION Network 168: Safety override - Clear AGTR3260_Toc_Do_AO
   RUNG wire#powerrail
      Contact( "PLC1_EStop_Latch" )
      wire#w1
      { S7_GenerateENO := "TRUE" } Move(in := 0.0, out1 => "AGTR3260_Toc_Do_AO")
   END_RUNG
   RUNG wire#powerrail
      Contact( "PLC1_Stop_Active" )
   END_RUNG wire#w1
   RUNG wire#powerrail
      Contact( "PLC1_Loi_Tong" )
   END_RUNG wire#w1
   // the same network as SCL:
   IF "PLC1_EStop_Latch" OR "PLC1_Stop_Active" OR "PLC1_Loi_Tong" THEN "AGTR3260_Toc_Do_AO" := 0.0; END_IF;
END_REGION

REGION Network 169: Safety override - Clear AGTR3260_Toc_Do_AO_Man
   RUNG wire#powerrail
      Contact( "PLC1_EStop_Latch" )
      wire#w1
      { S7_GenerateENO := "TRUE" } Move(in := 0.0, out1 => "AGTR3260_Toc_Do_AO_Man")
   END_RUNG
   RUNG wire#powerrail
      Contact( "PLC1_Stop_Active" )
   END_RUNG wire#w1
   RUNG wire#powerrail
      Contact( "PLC1_Loi_Tong" )
   END_RUNG wire#w1
   // the same network as SCL:
   IF "PLC1_EStop_Latch" OR "PLC1_Stop_Active" OR "PLC1_Loi_Tong" THEN
       "AGTR3260_Toc_Do_AO_Man" := 0.0;
   END_IF;
END_REGION

REGION Network 170: Safety override - Clear CV3206_Hoi_Bon2
   RUNG wire#powerrail
      Contact( "PLC1_EStop_Latch" )
      wire#w1
      { S7_GenerateENO := "TRUE" } Move(in := 0.0, out1 => "CV3206_Hoi_Bon2")
   END_RUNG
   RUNG wire#powerrail
      Contact( "PLC1_Stop_Active" )
   END_RUNG wire#w1
   RUNG wire#powerrail
      Contact( "PLC1_Loi_Tong" )
   END_RUNG wire#w1
   // the same network as SCL:
   IF "PLC1_EStop_Latch" OR "PLC1_Stop_Active" OR "PLC1_Loi_Tong" THEN "CV3206_Hoi_Bon2" := 0.0; END_IF;
END_REGION

REGION Network 171: Safety override - Clear CV3206_Hoi_Bon2_Man
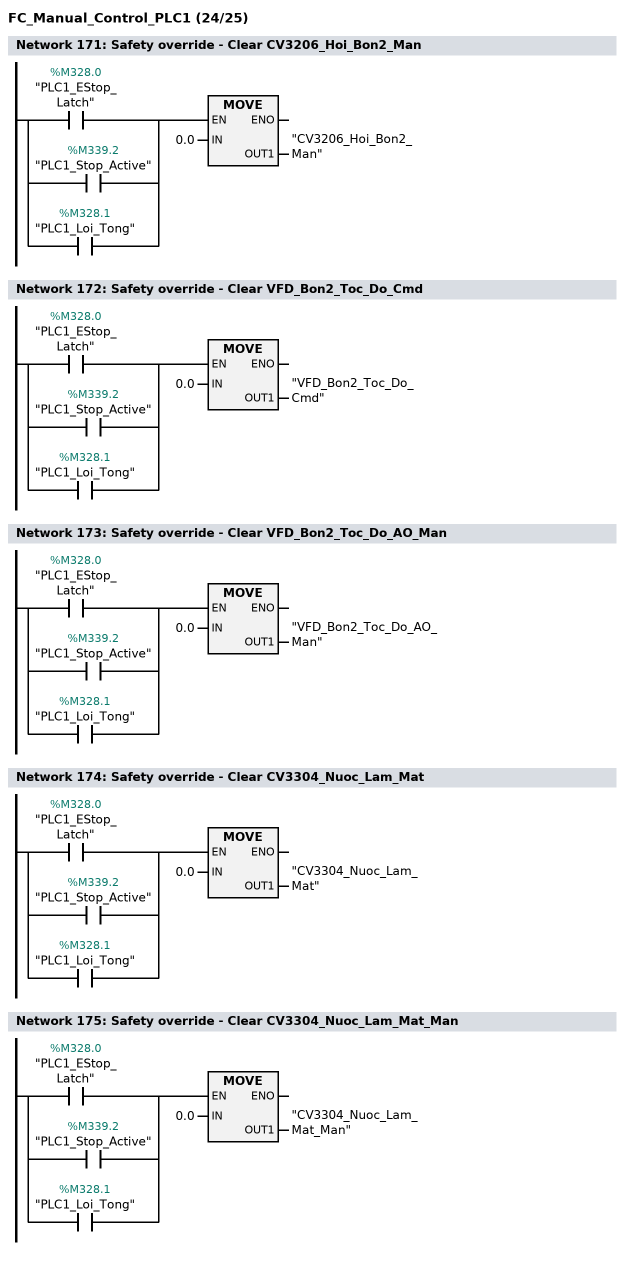
   RUNG wire#powerrail
      Contact( "PLC1_EStop_Latch" )
      wire#w1
      { S7_GenerateENO := "TRUE" } Move(in := 0.0, out1 => "CV3206_Hoi_Bon2_Man")
   END_RUNG
   RUNG wire#powerrail
      Contact( "PLC1_Stop_Active" )
   END_RUNG wire#w1
   RUNG wire#powerrail
      Contact( "PLC1_Loi_Tong" )
   END_RUNG wire#w1
   // the same network as SCL:
   IF "PLC1_EStop_Latch" OR "PLC1_Stop_Active" OR "PLC1_Loi_Tong" THEN "CV3206_Hoi_Bon2_Man" := 0.0; END_IF;
END_REGION

REGION Network 172: Safety override - Clear VFD_Bon2_Toc_Do_Cmd
   RUNG wire#powerrail
      Contact( "PLC1_EStop_Latch" )
      wire#w1
      { S7_GenerateENO := "TRUE" } Move(in := 0.0, out1 => "VFD_Bon2_Toc_Do_Cmd")
   END_RUNG
   RUNG wire#powerrail
      Contact( "PLC1_Stop_Active" )
   END_RUNG wire#w1
   RUNG wire#powerrail
      Contact( "PLC1_Loi_Tong" )
   END_RUNG wire#w1
   // the same network as SCL:
   IF "PLC1_EStop_Latch" OR "PLC1_Stop_Active" OR "PLC1_Loi_Tong" THEN "VFD_Bon2_Toc_Do_Cmd" := 0.0; END_IF;
END_REGION

REGION Network 173: Safety override - Clear VFD_Bon2_Toc_Do_AO_Man
   RUNG wire#powerrail
      Contact( "PLC1_EStop_Latch" )
      wire#w1
      { S7_GenerateENO := "TRUE" } Move(in := 0.0, out1 => "VFD_Bon2_Toc_Do_AO_Man")
   END_RUNG
   RUNG wire#powerrail
      Contact( "PLC1_Stop_Active" )
   END_RUNG wire#w1
   RUNG wire#powerrail
      Contact( "PLC1_Loi_Tong" )
   END_RUNG wire#w1
   // the same network as SCL:
   IF "PLC1_EStop_Latch" OR "PLC1_Stop_Active" OR "PLC1_Loi_Tong" THEN
       "VFD_Bon2_Toc_Do_AO_Man" := 0.0;
   END_IF;
END_REGION

REGION Network 174: Safety override - Clear CV3304_Nuoc_Lam_Mat
   RUNG wire#powerrail
      Contact( "PLC1_EStop_Latch" )
      wire#w1
      { S7_GenerateENO := "TRUE" } Move(in := 0.0, out1 => "CV3304_Nuoc_Lam_Mat")
   END_RUNG
   RUNG wire#powerrail
      Contact( "PLC1_Stop_Active" )
   END_RUNG wire#w1
   RUNG wire#powerrail
      Contact( "PLC1_Loi_Tong" )
   END_RUNG wire#w1
   // the same network as SCL:
   IF "PLC1_EStop_Latch" OR "PLC1_Stop_Active" OR "PLC1_Loi_Tong" THEN "CV3304_Nuoc_Lam_Mat" := 0.0; END_IF;
END_REGION

REGION Network 175: Safety override - Clear CV3304_Nuoc_Lam_Mat_Man
   RUNG wire#powerrail
      Contact( "PLC1_EStop_Latch" )
      wire#w1
      { S7_GenerateENO := "TRUE" } Move(in := 0.0, out1 => "CV3304_Nuoc_Lam_Mat_Man")
   END_RUNG
   RUNG wire#powerrail
      Contact( "PLC1_Stop_Active" )
   END_RUNG wire#w1
   RUNG wire#powerrail
      Contact( "PLC1_Loi_Tong" )
   END_RUNG wire#w1
   // the same network as SCL:
   IF "PLC1_EStop_Latch" OR "PLC1_Stop_Active" OR "PLC1_Loi_Tong" THEN
       "CV3304_Nuoc_Lam_Mat_Man" := 0.0;
   END_IF;
END_REGION

REGION Network 176: Safety override - Clear CV_Filler_Cap_Dich
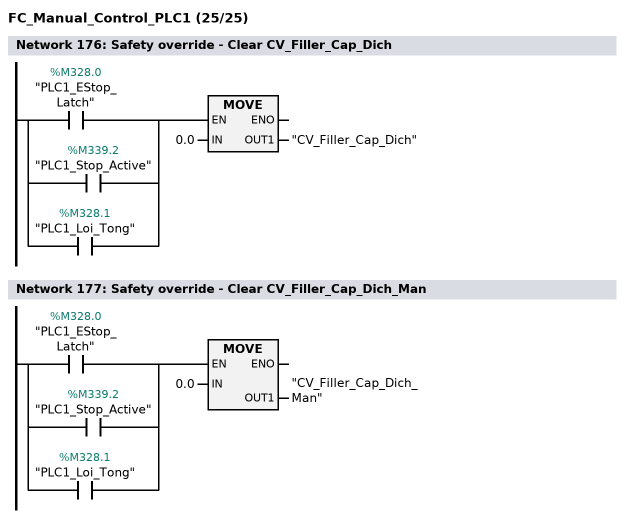
   RUNG wire#powerrail
      Contact( "PLC1_EStop_Latch" )
      wire#w1
      { S7_GenerateENO := "TRUE" } Move(in := 0.0, out1 => "CV_Filler_Cap_Dich")
   END_RUNG
   RUNG wire#powerrail
      Contact( "PLC1_Stop_Active" )
   END_RUNG wire#w1
   RUNG wire#powerrail
      Contact( "PLC1_Loi_Tong" )
   END_RUNG wire#w1
   // the same network as SCL:
   IF "PLC1_EStop_Latch" OR "PLC1_Stop_Active" OR "PLC1_Loi_Tong" THEN "CV_Filler_Cap_Dich" := 0.0; END_IF;
END_REGION

REGION Network 177: Safety override - Clear CV_Filler_Cap_Dich_Man
   RUNG wire#powerrail
      Contact( "PLC1_EStop_Latch" )
      wire#w1
      { S7_GenerateENO := "TRUE" } Move(in := 0.0, out1 => "CV_Filler_Cap_Dich_Man")
   END_RUNG
   RUNG wire#powerrail
      Contact( "PLC1_Stop_Active" )
   END_RUNG wire#w1
   RUNG wire#powerrail
      Contact( "PLC1_Loi_Tong" )
   END_RUNG wire#w1
   // the same network as SCL:
   IF "PLC1_EStop_Latch" OR "PLC1_Stop_Active" OR "PLC1_Loi_Tong" THEN
       "CV_Filler_Cap_Dich_Man" := 0.0;
   END_IF;
END_REGION
END_FUNCTION

FUNCTION "FC_VFD_Bon2_Hybrid" : Void   // FC70, LAD
{ S7_Optimized_Access := 'TRUE' }
VERSION : 0.1
// stored: AutoNumber true, IsIECCheckEnabled false, SetENOAutomatically false, UDAEnableTagReadback false
BEGIN

REGION Network 1: Điều khiển contactor VFD Bồn 2
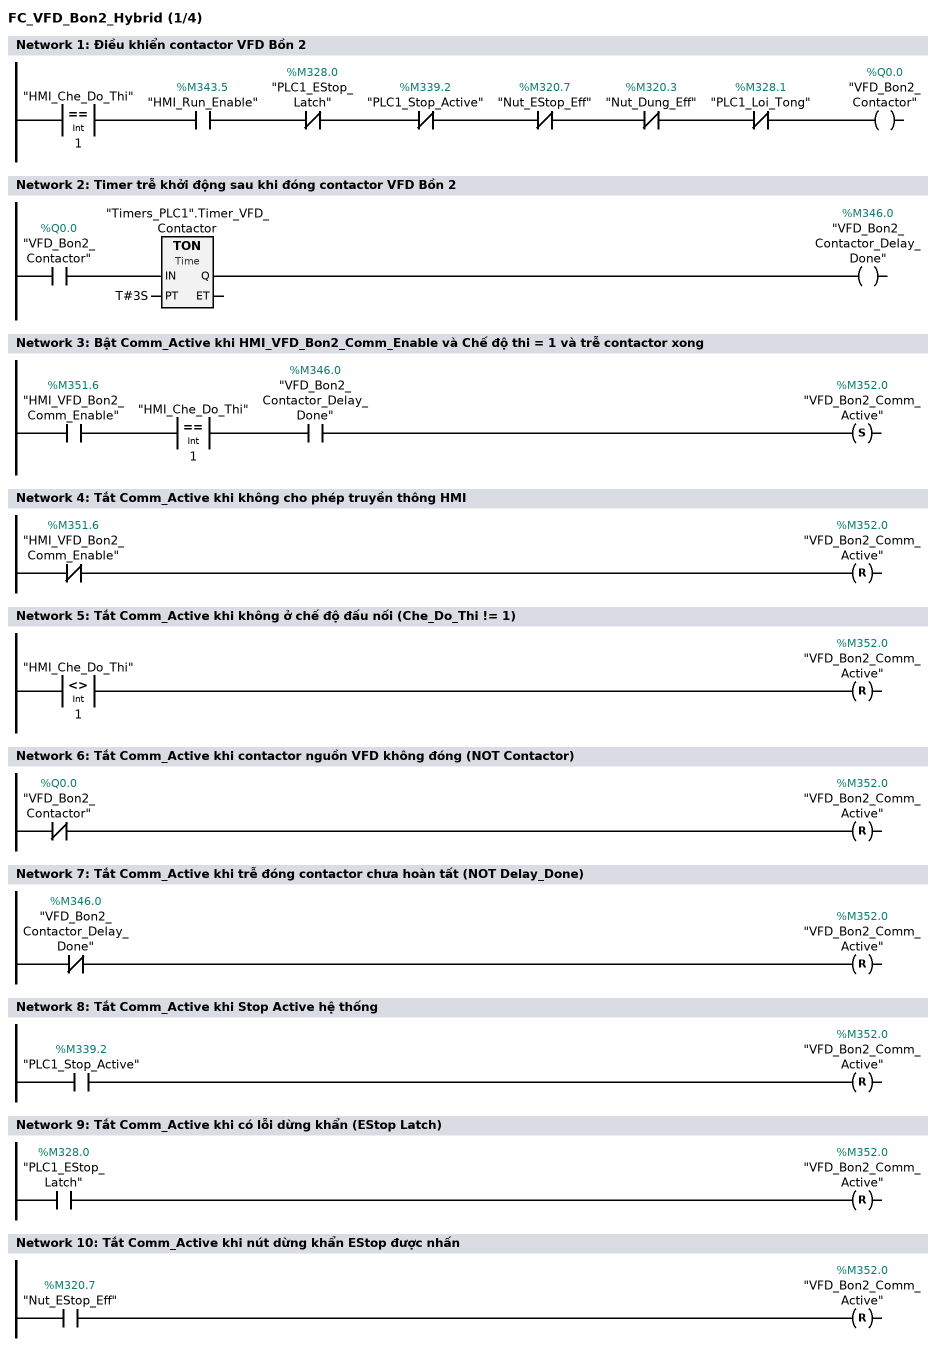
   RUNG wire#powerrail
      { S7_Templates := "SrcType := Int" } EQ_Contact(in1 := "HMI_Che_Do_Thi", in2 := 1)
      Contact( "HMI_Run_Enable" )
      I_Contact( "PLC1_EStop_Latch" )
      I_Contact( "PLC1_Stop_Active" )
      I_Contact( "Nut_EStop_Eff" )
      I_Contact( "Nut_Dung_Eff" )
      I_Contact( "PLC1_Loi_Tong" )
      Coil( "VFD_Bon2_Contactor" )
   END_RUNG
   // the same network as SCL:
   "VFD_Bon2_Contactor" := ("HMI_Che_Do_Thi" = 1) AND "HMI_Run_Enable" AND NOT "PLC1_EStop_Latch" AND NOT "PLC1_Stop_Active" AND NOT "Nut_EStop_Eff" AND NOT "Nut_Dung_Eff" AND NOT "PLC1_Loi_Tong";
END_REGION

REGION Network 2: Timer trễ khởi động sau khi đóng contactor VFD Bồn 2
   RUNG wire#powerrail
      Contact( "VFD_Bon2_Contactor" )
      { S7_Templates := "time_type := Time" } "Timers_PLC1".Timer_VFD_Contactor.TON(pt := T#3S, et =>)
      Coil( "VFD_Bon2_Contactor_Delay_Done" )
   END_RUNG
   // the same network as SCL:
   "Timers_PLC1".Timer_VFD_Contactor.TON(IN := "VFD_Bon2_Contactor", PT := T#3S);
   "VFD_Bon2_Contactor_Delay_Done" := "Timers_PLC1".Timer_VFD_Contactor.Q;
END_REGION

REGION Network 3: Bật Comm_Active khi HMI_VFD_Bon2_Comm_Enable và Chế độ thi = 1 và trễ contactor xong
   RUNG wire#powerrail
      Contact( "HMI_VFD_Bon2_Comm_Enable" )
      { S7_Templates := "SrcType := Int" } EQ_Contact(in1 := "HMI_Che_Do_Thi", in2 := 1)
      Contact( "VFD_Bon2_Contactor_Delay_Done" )
      S_Coil( "VFD_Bon2_Comm_Active" )
   END_RUNG
   // the same network as SCL:
   IF "HMI_VFD_Bon2_Comm_Enable" AND ("HMI_Che_Do_Thi" = 1) AND "VFD_Bon2_Contactor_Delay_Done" THEN
       "VFD_Bon2_Comm_Active" := TRUE;
   END_IF;
END_REGION

REGION Network 4: Tắt Comm_Active khi không cho phép truyền thông HMI
   RUNG wire#powerrail
      I_Contact( "HMI_VFD_Bon2_Comm_Enable" )
      R_Coil( "VFD_Bon2_Comm_Active" )
   END_RUNG
   // the same network as SCL:
   IF NOT "HMI_VFD_Bon2_Comm_Enable" THEN "VFD_Bon2_Comm_Active" := FALSE; END_IF;
END_REGION

REGION Network 5: Tắt Comm_Active khi không ở chế độ đấu nối (Che_Do_Thi != 1)
   RUNG wire#powerrail
      { S7_Templates := "SrcType := Int" } NE_Contact(in1 := "HMI_Che_Do_Thi", in2 := 1)
      R_Coil( "VFD_Bon2_Comm_Active" )
   END_RUNG
   // the same network as SCL:
   IF "HMI_Che_Do_Thi" <> 1 THEN "VFD_Bon2_Comm_Active" := FALSE; END_IF;
END_REGION

REGION Network 6: Tắt Comm_Active khi contactor nguồn VFD không đóng (NOT Contactor)
   RUNG wire#powerrail
      I_Contact( "VFD_Bon2_Contactor" )
      R_Coil( "VFD_Bon2_Comm_Active" )
   END_RUNG
   // the same network as SCL:
   IF NOT "VFD_Bon2_Contactor" THEN "VFD_Bon2_Comm_Active" := FALSE; END_IF;
END_REGION

REGION Network 7: Tắt Comm_Active khi trễ đóng contactor chưa hoàn tất (NOT Delay_Done)
   RUNG wire#powerrail
      I_Contact( "VFD_Bon2_Contactor_Delay_Done" )
      R_Coil( "VFD_Bon2_Comm_Active" )
   END_RUNG
   // the same network as SCL:
   IF NOT "VFD_Bon2_Contactor_Delay_Done" THEN "VFD_Bon2_Comm_Active" := FALSE; END_IF;
END_REGION

REGION Network 8: Tắt Comm_Active khi Stop Active hệ thống
   RUNG wire#powerrail
      Contact( "PLC1_Stop_Active" )
      R_Coil( "VFD_Bon2_Comm_Active" )
   END_RUNG
   // the same network as SCL:
   IF "PLC1_Stop_Active" THEN "VFD_Bon2_Comm_Active" := FALSE; END_IF;
END_REGION

REGION Network 9: Tắt Comm_Active khi có lỗi dừng khẩn (EStop Latch)
   RUNG wire#powerrail
      Contact( "PLC1_EStop_Latch" )
      R_Coil( "VFD_Bon2_Comm_Active" )
   END_RUNG
   // the same network as SCL:
   IF "PLC1_EStop_Latch" THEN "VFD_Bon2_Comm_Active" := FALSE; END_IF;
END_REGION

REGION Network 10: Tắt Comm_Active khi nút dừng khẩn EStop được nhấn
   RUNG wire#powerrail
      Contact( "Nut_EStop_Eff" )
      R_Coil( "VFD_Bon2_Comm_Active" )
   END_RUNG
   // the same network as SCL:
   IF "Nut_EStop_Eff" THEN "VFD_Bon2_Comm_Active" := FALSE; END_IF;
END_REGION

REGION Network 11: Tắt Comm_Active khi nút dừng hệ thống Stop được nhấn
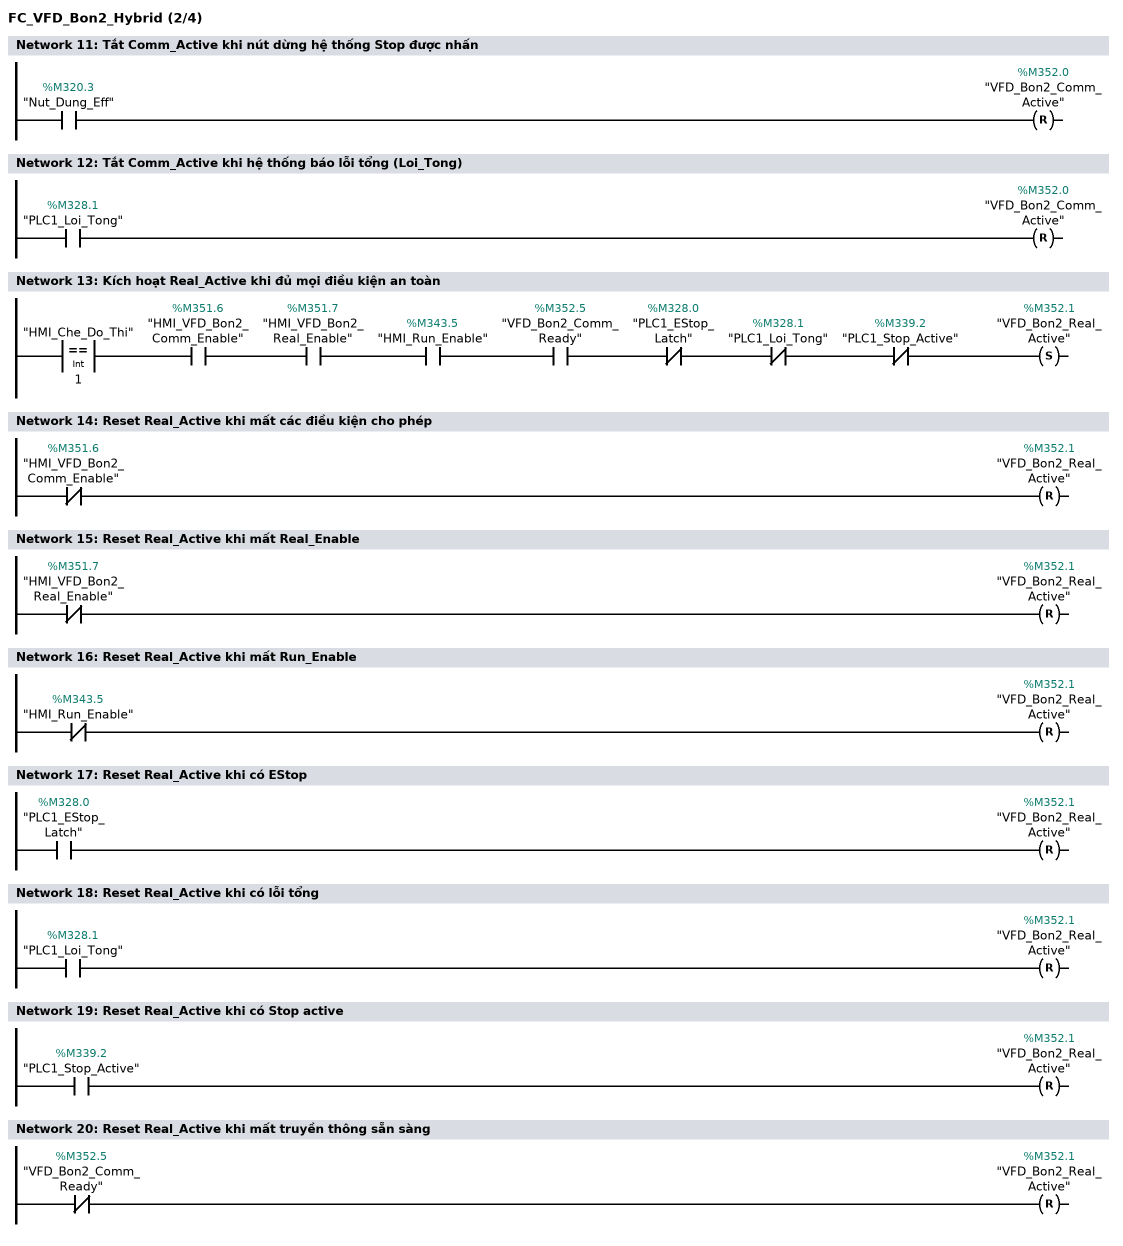
   RUNG wire#powerrail
      Contact( "Nut_Dung_Eff" )
      R_Coil( "VFD_Bon2_Comm_Active" )
   END_RUNG
   // the same network as SCL:
   IF "Nut_Dung_Eff" THEN "VFD_Bon2_Comm_Active" := FALSE; END_IF;
END_REGION

REGION Network 12: Tắt Comm_Active khi hệ thống báo lỗi tổng (Loi_Tong)
   RUNG wire#powerrail
      Contact( "PLC1_Loi_Tong" )
      R_Coil( "VFD_Bon2_Comm_Active" )
   END_RUNG
   // the same network as SCL:
   IF "PLC1_Loi_Tong" THEN "VFD_Bon2_Comm_Active" := FALSE; END_IF;
END_REGION

REGION Network 13: Kích hoạt Real_Active khi đủ mọi điều kiện an toàn
   RUNG wire#powerrail
      { S7_Templates := "SrcType := Int" } EQ_Contact(in1 := "HMI_Che_Do_Thi", in2 := 1)
      Contact( "HMI_VFD_Bon2_Comm_Enable" )
      Contact( "HMI_VFD_Bon2_Real_Enable" )
      Contact( "HMI_Run_Enable" )
      Contact( "VFD_Bon2_Comm_Ready" )
      I_Contact( "PLC1_EStop_Latch" )
      I_Contact( "PLC1_Loi_Tong" )
      I_Contact( "PLC1_Stop_Active" )
      S_Coil( "VFD_Bon2_Real_Active" )
   END_RUNG
   // the same network as SCL:
   IF ("HMI_Che_Do_Thi" = 1) AND "HMI_VFD_Bon2_Comm_Enable" AND "HMI_VFD_Bon2_Real_Enable" AND "HMI_Run_Enable" AND "VFD_Bon2_Comm_Ready" AND NOT "PLC1_EStop_Latch" AND NOT "PLC1_Loi_Tong" AND NOT "PLC1_Stop_Active" THEN
       "VFD_Bon2_Real_Active" := TRUE;
   END_IF;
END_REGION

REGION Network 14: Reset Real_Active khi mất các điều kiện cho phép
   RUNG wire#powerrail
      I_Contact( "HMI_VFD_Bon2_Comm_Enable" )
      R_Coil( "VFD_Bon2_Real_Active" )
   END_RUNG
   // the same network as SCL:
   IF NOT "HMI_VFD_Bon2_Comm_Enable" THEN "VFD_Bon2_Real_Active" := FALSE; END_IF;
END_REGION

REGION Network 15: Reset Real_Active khi mất Real_Enable
   RUNG wire#powerrail
      I_Contact( "HMI_VFD_Bon2_Real_Enable" )
      R_Coil( "VFD_Bon2_Real_Active" )
   END_RUNG
   // the same network as SCL:
   IF NOT "HMI_VFD_Bon2_Real_Enable" THEN "VFD_Bon2_Real_Active" := FALSE; END_IF;
END_REGION

REGION Network 16: Reset Real_Active khi mất Run_Enable
   RUNG wire#powerrail
      I_Contact( "HMI_Run_Enable" )
      R_Coil( "VFD_Bon2_Real_Active" )
   END_RUNG
   // the same network as SCL:
   IF NOT "HMI_Run_Enable" THEN "VFD_Bon2_Real_Active" := FALSE; END_IF;
END_REGION

REGION Network 17: Reset Real_Active khi có EStop
   RUNG wire#powerrail
      Contact( "PLC1_EStop_Latch" )
      R_Coil( "VFD_Bon2_Real_Active" )
   END_RUNG
   // the same network as SCL:
   IF "PLC1_EStop_Latch" THEN "VFD_Bon2_Real_Active" := FALSE; END_IF;
END_REGION

REGION Network 18: Reset Real_Active khi có lỗi tổng
   RUNG wire#powerrail
      Contact( "PLC1_Loi_Tong" )
      R_Coil( "VFD_Bon2_Real_Active" )
   END_RUNG
   // the same network as SCL:
   IF "PLC1_Loi_Tong" THEN "VFD_Bon2_Real_Active" := FALSE; END_IF;
END_REGION

REGION Network 19: Reset Real_Active khi có Stop active
   RUNG wire#powerrail
      Contact( "PLC1_Stop_Active" )
      R_Coil( "VFD_Bon2_Real_Active" )
   END_RUNG
   // the same network as SCL:
   IF "PLC1_Stop_Active" THEN "VFD_Bon2_Real_Active" := FALSE; END_IF;
END_REGION

REGION Network 20: Reset Real_Active khi mất truyền thông sẵn sàng
   RUNG wire#powerrail
      I_Contact( "VFD_Bon2_Comm_Ready" )
      R_Coil( "VFD_Bon2_Real_Active" )
   END_RUNG
   // the same network as SCL:
   IF NOT "VFD_Bon2_Comm_Ready" THEN "VFD_Bon2_Real_Active" := FALSE; END_IF;
END_REGION

REGION Network 21: Reset Real_Active khi không ở chế độ đấu nối
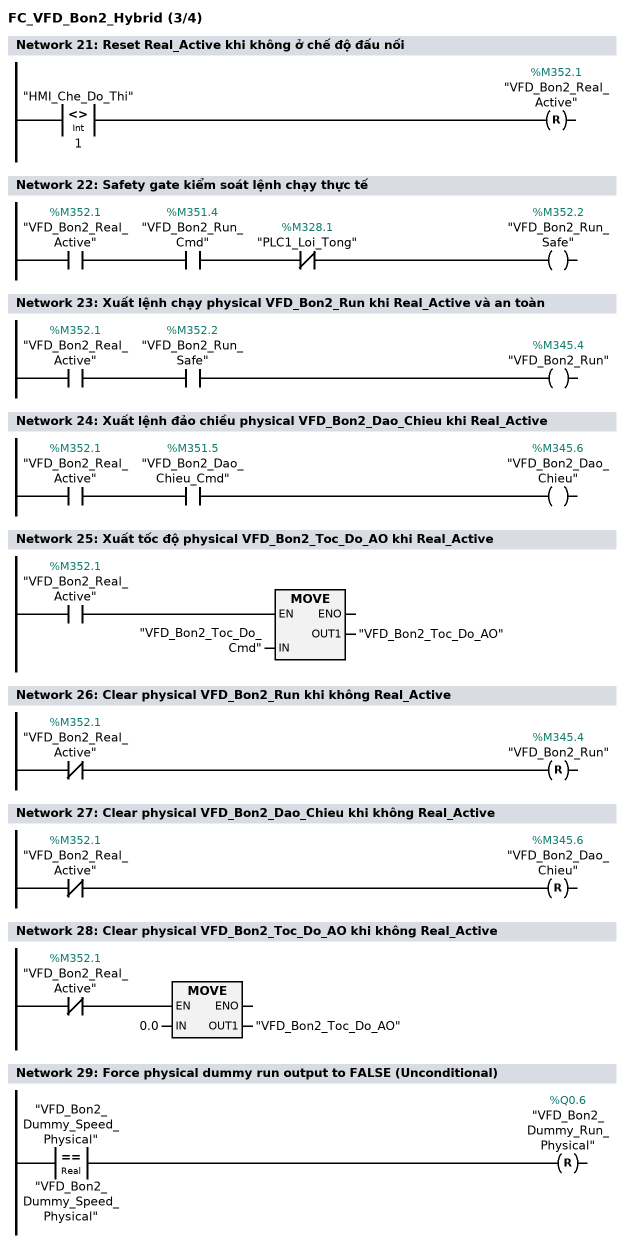
   RUNG wire#powerrail
      { S7_Templates := "SrcType := Int" } NE_Contact(in1 := "HMI_Che_Do_Thi", in2 := 1)
      R_Coil( "VFD_Bon2_Real_Active" )
   END_RUNG
   // the same network as SCL:
   IF "HMI_Che_Do_Thi" <> 1 THEN "VFD_Bon2_Real_Active" := FALSE; END_IF;
END_REGION

REGION Network 22: Safety gate kiểm soát lệnh chạy thực tế
   RUNG wire#powerrail
      Contact( "VFD_Bon2_Real_Active" )
      Contact( "VFD_Bon2_Run_Cmd" )
      I_Contact( "PLC1_Loi_Tong" )
      Coil( "VFD_Bon2_Run_Safe" )
   END_RUNG
   // the same network as SCL:
   "VFD_Bon2_Run_Safe" := "VFD_Bon2_Real_Active" AND "VFD_Bon2_Run_Cmd" AND NOT "PLC1_Loi_Tong";
END_REGION

REGION Network 23: Xuất lệnh chạy physical VFD_Bon2_Run khi Real_Active và an toàn
   RUNG wire#powerrail
      Contact( "VFD_Bon2_Real_Active" )
      Contact( "VFD_Bon2_Run_Safe" )
      Coil( "VFD_Bon2_Run" )
   END_RUNG
   // the same network as SCL:
   "VFD_Bon2_Run" := "VFD_Bon2_Real_Active" AND "VFD_Bon2_Run_Safe";
END_REGION

REGION Network 24: Xuất lệnh đảo chiều physical VFD_Bon2_Dao_Chieu khi Real_Active
   RUNG wire#powerrail
      Contact( "VFD_Bon2_Real_Active" )
      Contact( "VFD_Bon2_Dao_Chieu_Cmd" )
      Coil( "VFD_Bon2_Dao_Chieu" )
   END_RUNG
   // the same network as SCL:
   "VFD_Bon2_Dao_Chieu" := "VFD_Bon2_Real_Active" AND "VFD_Bon2_Dao_Chieu_Cmd";
END_REGION

REGION Network 25: Xuất tốc độ physical VFD_Bon2_Toc_Do_AO khi Real_Active
   RUNG wire#powerrail
      Contact( "VFD_Bon2_Real_Active" )
      { S7_GenerateENO := "TRUE" } Move(in := "VFD_Bon2_Toc_Do_Cmd", out1 => "VFD_Bon2_Toc_Do_AO")
   END_RUNG
   // the same network as SCL:
   IF "VFD_Bon2_Real_Active" THEN "VFD_Bon2_Toc_Do_AO" := "VFD_Bon2_Toc_Do_Cmd"; END_IF;
END_REGION

REGION Network 26: Clear physical VFD_Bon2_Run khi không Real_Active
   RUNG wire#powerrail
      I_Contact( "VFD_Bon2_Real_Active" )
      R_Coil( "VFD_Bon2_Run" )
   END_RUNG
   // the same network as SCL:
   IF NOT "VFD_Bon2_Real_Active" THEN "VFD_Bon2_Run" := FALSE; END_IF;
END_REGION

REGION Network 27: Clear physical VFD_Bon2_Dao_Chieu khi không Real_Active
   RUNG wire#powerrail
      I_Contact( "VFD_Bon2_Real_Active" )
      R_Coil( "VFD_Bon2_Dao_Chieu" )
   END_RUNG
   // the same network as SCL:
   IF NOT "VFD_Bon2_Real_Active" THEN "VFD_Bon2_Dao_Chieu" := FALSE; END_IF;
END_REGION

REGION Network 28: Clear physical VFD_Bon2_Toc_Do_AO khi không Real_Active
   RUNG wire#powerrail
      I_Contact( "VFD_Bon2_Real_Active" )
      { S7_GenerateENO := "TRUE" } Move(in := 0.0, out1 => "VFD_Bon2_Toc_Do_AO")
   END_RUNG
   // the same network as SCL:
   IF NOT "VFD_Bon2_Real_Active" THEN "VFD_Bon2_Toc_Do_AO" := 0.0; END_IF;
END_REGION

REGION Network 29: Force physical dummy run output to FALSE (Unconditional)
   RUNG wire#powerrail
      { S7_Templates := "SrcType := Real" } EQ_Contact(in1 := "VFD_Bon2_Dummy_Speed_Physical", in2 := "VFD_Bon2_Dummy_Speed_Physical")
      R_Coil( "VFD_Bon2_Dummy_Run_Physical" )
   END_RUNG
   // the same network as SCL:
   IF "VFD_Bon2_Dummy_Speed_Physical" = "VFD_Bon2_Dummy_Speed_Physical" THEN
       "VFD_Bon2_Dummy_Run_Physical" := FALSE;
   END_IF;
END_REGION

REGION Network 30: Force physical dummy reverse output to FALSE (Unconditional)
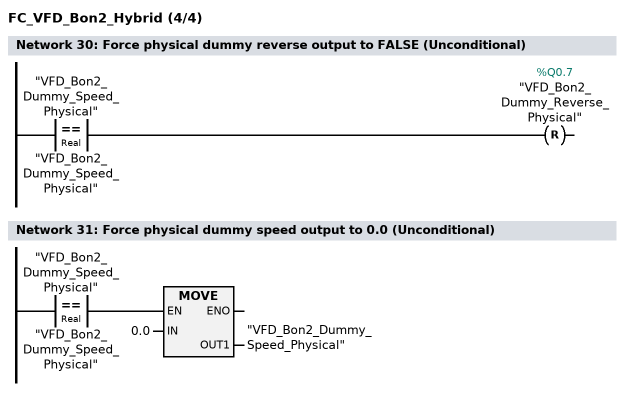
   RUNG wire#powerrail
      { S7_Templates := "SrcType := Real" } EQ_Contact(in1 := "VFD_Bon2_Dummy_Speed_Physical", in2 := "VFD_Bon2_Dummy_Speed_Physical")
      R_Coil( "VFD_Bon2_Dummy_Reverse_Physical" )
   END_RUNG
   // the same network as SCL:
   IF "VFD_Bon2_Dummy_Speed_Physical" = "VFD_Bon2_Dummy_Speed_Physical" THEN
       "VFD_Bon2_Dummy_Reverse_Physical" := FALSE;
   END_IF;
END_REGION

REGION Network 31: Force physical dummy speed output to 0.0 (Unconditional)
   RUNG wire#powerrail
      { S7_Templates := "SrcType := Real" } EQ_Contact(in1 := "VFD_Bon2_Dummy_Speed_Physical", in2 := "VFD_Bon2_Dummy_Speed_Physical")
      { S7_GenerateENO := "TRUE" } Move(in := 0.0, out1 => "VFD_Bon2_Dummy_Speed_Physical")
   END_RUNG
   // the same network as SCL:
   IF "VFD_Bon2_Dummy_Speed_Physical" = "VFD_Bon2_Dummy_Speed_Physical" THEN
       "VFD_Bon2_Dummy_Speed_Physical" := 0.0;
   END_IF;
END_REGION
END_FUNCTION

FUNCTION "FC_HMI_Mirror_PLC1" : Void   // FC40, LAD
{ S7_Optimized_Access := 'TRUE' }
VERSION : 0.1
// stored: AutoNumber true, IsIECCheckEnabled false, SetENOAutomatically false, UDAEnableTagReadback false
BEGIN

REGION Network 1: Mirror VFD_Bon2_Contactor
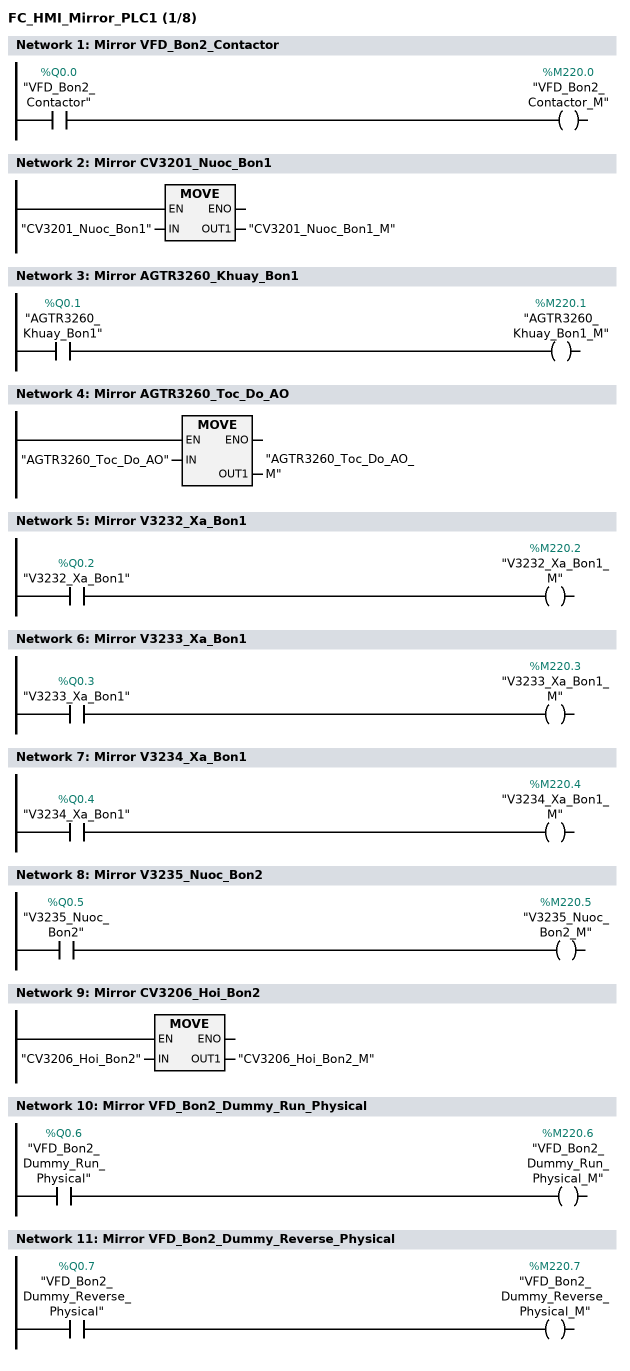
   RUNG wire#powerrail
      Contact( "VFD_Bon2_Contactor" )
      Coil( "VFD_Bon2_Contactor_M" )
   END_RUNG
   // the same network as SCL:
   "VFD_Bon2_Contactor_M" := "VFD_Bon2_Contactor";
END_REGION

REGION Network 2: Mirror CV3201_Nuoc_Bon1
   RUNG wire#powerrail
      { S7_GenerateENO := "TRUE" } Move(in := "CV3201_Nuoc_Bon1", out1 => "CV3201_Nuoc_Bon1_M")
   END_RUNG
   // the same network as SCL:
   "CV3201_Nuoc_Bon1_M" := "CV3201_Nuoc_Bon1";
END_REGION

REGION Network 3: Mirror AGTR3260_Khuay_Bon1
   RUNG wire#powerrail
      Contact( "AGTR3260_Khuay_Bon1" )
      Coil( "AGTR3260_Khuay_Bon1_M" )
   END_RUNG
   // the same network as SCL:
   "AGTR3260_Khuay_Bon1_M" := "AGTR3260_Khuay_Bon1";
END_REGION

REGION Network 4: Mirror AGTR3260_Toc_Do_AO
   RUNG wire#powerrail
      { S7_GenerateENO := "TRUE" } Move(in := "AGTR3260_Toc_Do_AO", out1 => "AGTR3260_Toc_Do_AO_M")
   END_RUNG
   // the same network as SCL:
   "AGTR3260_Toc_Do_AO_M" := "AGTR3260_Toc_Do_AO";
END_REGION

REGION Network 5: Mirror V3232_Xa_Bon1
   RUNG wire#powerrail
      Contact( "V3232_Xa_Bon1" )
      Coil( "V3232_Xa_Bon1_M" )
   END_RUNG
   // the same network as SCL:
   "V3232_Xa_Bon1_M" := "V3232_Xa_Bon1";
END_REGION

REGION Network 6: Mirror V3233_Xa_Bon1
   RUNG wire#powerrail
      Contact( "V3233_Xa_Bon1" )
      Coil( "V3233_Xa_Bon1_M" )
   END_RUNG
   // the same network as SCL:
   "V3233_Xa_Bon1_M" := "V3233_Xa_Bon1";
END_REGION

REGION Network 7: Mirror V3234_Xa_Bon1
   RUNG wire#powerrail
      Contact( "V3234_Xa_Bon1" )
      Coil( "V3234_Xa_Bon1_M" )
   END_RUNG
   // the same network as SCL:
   "V3234_Xa_Bon1_M" := "V3234_Xa_Bon1";
END_REGION

REGION Network 8: Mirror V3235_Nuoc_Bon2
   RUNG wire#powerrail
      Contact( "V3235_Nuoc_Bon2" )
      Coil( "V3235_Nuoc_Bon2_M" )
   END_RUNG
   // the same network as SCL:
   "V3235_Nuoc_Bon2_M" := "V3235_Nuoc_Bon2";
END_REGION

REGION Network 9: Mirror CV3206_Hoi_Bon2
   RUNG wire#powerrail
      { S7_GenerateENO := "TRUE" } Move(in := "CV3206_Hoi_Bon2", out1 => "CV3206_Hoi_Bon2_M")
   END_RUNG
   // the same network as SCL:
   "CV3206_Hoi_Bon2_M" := "CV3206_Hoi_Bon2";
END_REGION

REGION Network 10: Mirror VFD_Bon2_Dummy_Run_Physical
   RUNG wire#powerrail
      Contact( "VFD_Bon2_Dummy_Run_Physical" )
      Coil( "VFD_Bon2_Dummy_Run_Physical_M" )
   END_RUNG
   // the same network as SCL:
   "VFD_Bon2_Dummy_Run_Physical_M" := "VFD_Bon2_Dummy_Run_Physical";
END_REGION

REGION Network 11: Mirror VFD_Bon2_Dummy_Reverse_Physical
   RUNG wire#powerrail
      Contact( "VFD_Bon2_Dummy_Reverse_Physical" )
      Coil( "VFD_Bon2_Dummy_Reverse_Physical_M" )
   END_RUNG
   // the same network as SCL:
   "VFD_Bon2_Dummy_Reverse_Physical_M" := "VFD_Bon2_Dummy_Reverse_Physical";
END_REGION

REGION Network 12: Mirror VFD_Bon2_Dummy_Speed_Physical
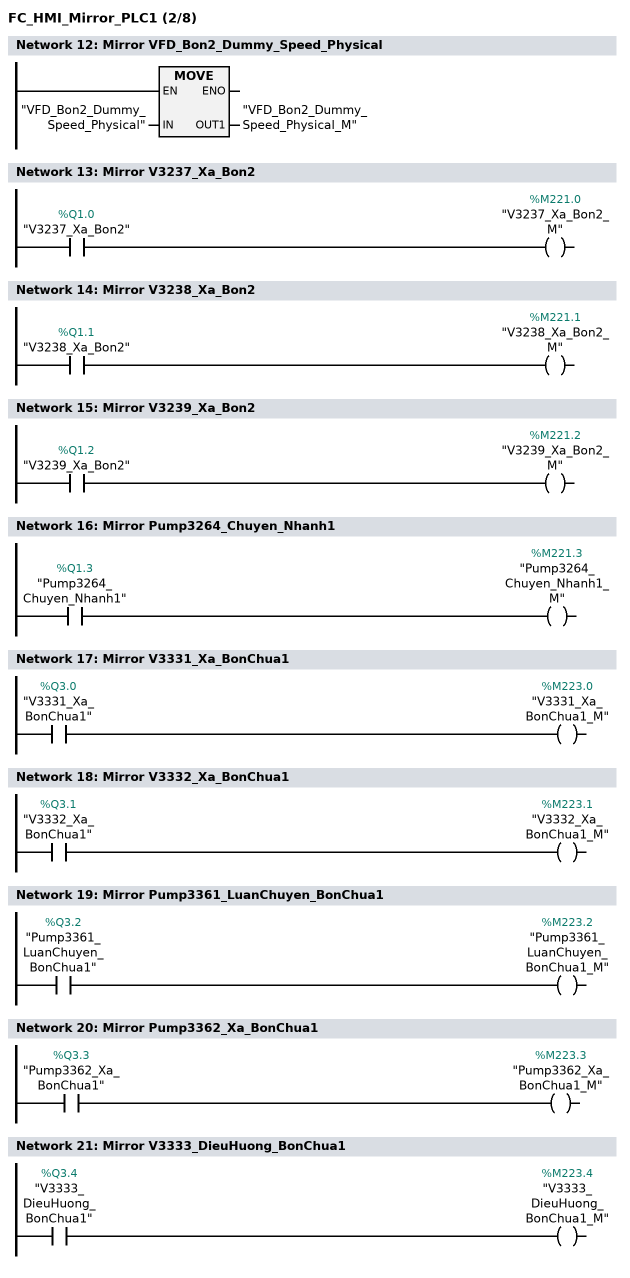
   RUNG wire#powerrail
      { S7_GenerateENO := "TRUE" } Move(in := "VFD_Bon2_Dummy_Speed_Physical", out1 => "VFD_Bon2_Dummy_Speed_Physical_M")
   END_RUNG
   // the same network as SCL:
   "VFD_Bon2_Dummy_Speed_Physical_M" := "VFD_Bon2_Dummy_Speed_Physical";
END_REGION

REGION Network 13: Mirror V3237_Xa_Bon2
   RUNG wire#powerrail
      Contact( "V3237_Xa_Bon2" )
      Coil( "V3237_Xa_Bon2_M" )
   END_RUNG
   // the same network as SCL:
   "V3237_Xa_Bon2_M" := "V3237_Xa_Bon2";
END_REGION

REGION Network 14: Mirror V3238_Xa_Bon2
   RUNG wire#powerrail
      Contact( "V3238_Xa_Bon2" )
      Coil( "V3238_Xa_Bon2_M" )
   END_RUNG
   // the same network as SCL:
   "V3238_Xa_Bon2_M" := "V3238_Xa_Bon2";
END_REGION

REGION Network 15: Mirror V3239_Xa_Bon2
   RUNG wire#powerrail
      Contact( "V3239_Xa_Bon2" )
      Coil( "V3239_Xa_Bon2_M" )
   END_RUNG
   // the same network as SCL:
   "V3239_Xa_Bon2_M" := "V3239_Xa_Bon2";
END_REGION

REGION Network 16: Mirror Pump3264_Chuyen_Nhanh1
   RUNG wire#powerrail
      Contact( "Pump3264_Chuyen_Nhanh1" )
      Coil( "Pump3264_Chuyen_Nhanh1_M" )
   END_RUNG
   // the same network as SCL:
   "Pump3264_Chuyen_Nhanh1_M" := "Pump3264_Chuyen_Nhanh1";
END_REGION

REGION Network 17: Mirror V3331_Xa_BonChua1
   RUNG wire#powerrail
      Contact( "V3331_Xa_BonChua1" )
      Coil( "V3331_Xa_BonChua1_M" )
   END_RUNG
   // the same network as SCL:
   "V3331_Xa_BonChua1_M" := "V3331_Xa_BonChua1";
END_REGION

REGION Network 18: Mirror V3332_Xa_BonChua1
   RUNG wire#powerrail
      Contact( "V3332_Xa_BonChua1" )
      Coil( "V3332_Xa_BonChua1_M" )
   END_RUNG
   // the same network as SCL:
   "V3332_Xa_BonChua1_M" := "V3332_Xa_BonChua1";
END_REGION

REGION Network 19: Mirror Pump3361_LuanChuyen_BonChua1
   RUNG wire#powerrail
      Contact( "Pump3361_LuanChuyen_BonChua1" )
      Coil( "Pump3361_LuanChuyen_BonChua1_M" )
   END_RUNG
   // the same network as SCL:
   "Pump3361_LuanChuyen_BonChua1_M" := "Pump3361_LuanChuyen_BonChua1";
END_REGION

REGION Network 20: Mirror Pump3362_Xa_BonChua1
   RUNG wire#powerrail
      Contact( "Pump3362_Xa_BonChua1" )
      Coil( "Pump3362_Xa_BonChua1_M" )
   END_RUNG
   // the same network as SCL:
   "Pump3362_Xa_BonChua1_M" := "Pump3362_Xa_BonChua1";
END_REGION

REGION Network 21: Mirror V3333_DieuHuong_BonChua1
   RUNG wire#powerrail
      Contact( "V3333_DieuHuong_BonChua1" )
      Coil( "V3333_DieuHuong_BonChua1_M" )
   END_RUNG
   // the same network as SCL:
   "V3333_DieuHuong_BonChua1_M" := "V3333_DieuHuong_BonChua1";
END_REGION

REGION Network 22: Mirror V3334_DieuHuong_BonChua1
